GVL_1.Setpoint_M_Belts:=Setpoint_Belts_TOP_IN;
GVL_1.Setpoint_Belt_Feeder:=Setpoint_M_Belt_Feeder_IN;
GVL_1.Setpoint_SteamFan:=Setpoint_SteamFan_IN;
GVL_1.Setpoint_Compressor:=Setpoint_Compressor_IN;
GVL_1.Ps_202_out:=Ps_202;
GVL_1.Ps_203_out:=Ps_203;
GVL_1.volFracAir202_out:=volFracAir202;
GVL_1.volFracAir203_out:=volFracAir203;
GVL_1.volFracAirO2_out:=volFracAirO2;






IF SteamFAN_Switch_ON_manu AND SteamFan_ON_manu AND  Setpoint_SteamFan_Visu  >20.0 THEN
OK_For_HEAT_WHILE_FAN_IS_ON:=TRUE;
ELSE
OK_For_HEAT_WHILE_FAN_IS_ON:=FALSE;
END_IF;

END_PROGRAM

// ---- POUs/FB_Blink.TcPOU
FUNCTION_BLOCK FB_Blink
VAR_INPUT
	bStart:BOOL;
	tTakt:TIME:=t#0.5s;
END_VAR
VAR_OUTPUT
	bBlink:BOOL;
END_VAR
VAR
	fbT1:TON;
	fbT2:TON;
END_VAR

(*erste Hälfte der Blinkperiode, FB-Aufruf und Beschaltung in einem *)
fbT1(IN:=bStart AND NOT fbt2.Q,
	PT:= tTakt/2,
	Q=> bBlink,
	ET=> );


(*zweite Hälfte der Blinkperiode; Bsp. programmiert mit getrennter Beschaltung und Aufruf*)

fbt2.IN := fbT1.Q;   		(*vorheriges Beschalten der InputVar*)
fbt2.PT := tTakt / 2;  	(*vorheriges Beschalten der InputVar*)

fbT2();  					(*eigentliche FB-Instanz-Aufruf*)

END_FUNCTION_BLOCK

// ---- POUs/Average.TcPOU
FUNCTION_BLOCK Average
VAR_INPUT
	Input_AV: REAL;
END_VAR
VAR_OUTPUT
	OUTPUT_AV:REAL;
END_VAR
VAR
	C_AV: INT;
	summary_AV: REAL;
END_VAR



CASE C_AV OF


0:summary_AV:=0;	C_AV:=1;
1:summary_AV:=Input_AV;	C_AV:=2;
2:summary_AV:=summary_AV+Input_AV; C_AV:=3;
3:summary_AV:=summary_AV+Input_AV; C_AV:=4;
4:summary_AV:=summary_AV+Input_AV; C_AV:=5;
5:summary_AV:=summary_AV+Input_AV; C_AV:=6;
6:summary_AV:=summary_AV+Input_AV; C_AV:=7;
7:summary_AV:=summary_AV+Input_AV; C_AV:=8;
8:summary_AV:=summary_AV+Input_AV; C_AV:=9;
9:summary_AV:=summary_AV+Input_AV; C_AV:=10;
10:summary_AV:=summary_AV+Input_AV; C_AV:=11;
11:summary_AV:=summary_AV+Input_AV; C_AV:=12;
12:summary_AV:=summary_AV+Input_AV; C_AV:=13;
13:summary_AV:=summary_AV+Input_AV; C_AV:=14;
14:summary_AV:=summary_AV+Input_AV; C_AV:=15;
15:summary_AV:=summary_AV+Input_AV; C_AV:=16;
16:summary_AV:=summary_AV+Input_AV; C_AV:=17;
17:summary_AV:=summary_AV+Input_AV; C_AV:=18;
18:summary_AV:=summary_AV+Input_AV; C_AV:=19;
19:summary_AV:=summary_AV+Input_AV; C_AV:=20;
20:summary_AV:=summary_AV+Input_AV; C_AV:=21;
21:summary_AV:=summary_AV+Input_AV; C_AV:=22;
22:summary_AV:=summary_AV+Input_AV; C_AV:=23;
23:summary_AV:=summary_AV+Input_AV; C_AV:=24;
24:summary_AV:=summary_AV+Input_AV; C_AV:=25;
25:summary_AV:=summary_AV+Input_AV; C_AV:=26;
26:summary_AV:=summary_AV+Input_AV; C_AV:=27;
27:summary_AV:=summary_AV+Input_AV; C_AV:=28;
28:summary_AV:=summary_AV+Input_AV; C_AV:=29;
29:summary_AV:=summary_AV+Input_AV; C_AV:=30;
30:summary_AV:=summary_AV+Input_AV; C_AV:=31;
31:summary_AV:=summary_AV+Input_AV; C_AV:=32;
32:summary_AV:=summary_AV+Input_AV; C_AV:=33;
33:summary_AV:=summary_AV+Input_AV; C_AV:=34;
34:summary_AV:=summary_AV+Input_AV; C_AV:=35;
35:summary_AV:=summary_AV+Input_AV; C_AV:=36;
36:summary_AV:=summary_AV+Input_AV; C_AV:=37;
37:summary_AV:=summary_AV+Input_AV; C_AV:=38;
38:summary_AV:=summary_AV+Input_AV; C_AV:=39;
39:summary_AV:=summary_AV+Input_AV; C_AV:=40;
40:summary_AV:=summary_AV+Input_AV; C_AV:=41;
41:summary_AV:=summary_AV+Input_AV; C_AV:=42;
42:summary_AV:=summary_AV+Input_AV; C_AV:=43;
43:summary_AV:=summary_AV+Input_AV; C_AV:=44;
44:summary_AV:=summary_AV+Input_AV; C_AV:=45;
45:summary_AV:=summary_AV+Input_AV; C_AV:=46;
46:summary_AV:=summary_AV+Input_AV; C_AV:=47;
47:summary_AV:=summary_AV+Input_AV; C_AV:=48;
48:summary_AV:=summary_AV+Input_AV; C_AV:=49;
49:summary_AV:=summary_AV+Input_AV; C_AV:=50;
50:summary_AV:=summary_AV+Input_AV; C_AV:=51;
51:OUTPUT_AV:=summary_AV/50.0; C_AV:=0;

END_CASE

END_FUNCTION_BLOCK

// ---- POUs/Meine_HYST.TcPOU
FUNCTION_BLOCK Meine_HYST
VAR_INPUT
	Hyst_Value: INT;
	Hyst_Low_Limit: INT;
	Hyst_Hight_Limit: INT;
END_VAR
VAR_OUTPUT
	Hyst_OUT:BOOL ;
END_VAR
VAR
(*ZEITEN*)

	TON1:TON;
	IN_T1:BOOL;
	OUT_T1:BOOL;
	TON2:TON;
	IN_T2:BOOL;
	OUT_T2:BOOL;



END_VAR




(*Hyterese Universell für Heizmatten*)

IF Hyst_Value < Hyst_Low_Limit  THEN IN_T1:=TRUE; ELSE IF Hyst_Value  >= Hyst_Hight_Limit   THEN IN_T1:=FALSE; END_IF END_IF
IF OUT_T1 THEN Hyst_OUT:=TRUE; ELSE Hyst_OUT:=FALSE; END_IF



TON1(IN:=IN_T1 , PT:=t#30s, Q=>OUT_T1 , ET=> ); (*ZEIT Hauptschütz einschalten*)

TON2(IN:=IN_T2 , PT:=t#30s, Q=>OUT_T2 , ET=> ); (*ZEIT Überwachung Hauptschütz einschalten*)

END_FUNCTION_BLOCK

// ---- POUs/Controller.TcPOU
FUNCTION_BLOCK Controller
VAR_INPUT
END_VAR
VAR_OUTPUT
END_VAR
VAR
	CTRL_1: FB_BasicPID;
	CTRL_2: FB_BasicPID;
	
	Heat_REG1_CTRL:CTRL_PID;
	Heat_REG2_CTRL:CTRL_PID;
	Heat_REG3_CTRL:CTRL_PID;
	Heat_REG4_CTRL:CTRL_PID;
	Heat_REG5_CTRL:CTRL_PID;
	Heat_REG6_CTRL:CTRL_PID;
	Heat_REG7_CTRL:CTRL_PID;
	Heat_REG8_CTRL:CTRL_PID;
	
	
	
	Heat_REG1_PWM:CTRL_PWM;
	Heat_REG2_PWM:CTRL_PWM;
	Heat_REG3_PWM:CTRL_PWM;
	Heat_REG4_PWM:CTRL_PWM;
	Heat_REG5_PWM:CTRL_PWM;
	Heat_REG6_PWM:CTRL_PWM;
	Heat_REG7_PWM:CTRL_PWM;
	Heat_REG8_PWM:CTRL_PWM;
	
	
	
	
	
	fPWMDutyCycle1_out: REAL;
	fPWMDutyCycle2_out: REAL;
	fPWMDutyCycle3_out: REAL;
	fPWMDutyCycle4_out: REAL;
	
	
	
	
	
	HEAT_Reg_2_OUT_local: BOOL;
	HEAT_Reg_1_OUT_local: BOOL;
	HEAT_Reg_3_OUT_local: BOOL;
END_VAR





(* Infos zu den Reglern:

1. Es wurde eine von OSCAT-entwickelte Library-Sammlung zusammengefasst, damit diese auch als-FB/FC-Sammlung direkt im TC3-eingebunden werden können.
Die direkte Einbindung der OSCAT-Libs im Lib-Repository von TC3 macht Probleme, desshalb die direkte FB/FC Sammlung

In dieser Sammlung (Ornder PID_Controller_LIB) sind die CRT_PID & CTRL_PWM von OSCAT enthalten, welche für die Heizregler im Fall TRISS eingesetzt werden.

Wichtig als Backround: Die Controller_LIbs von Beckhoff sind etwas teuer, wenn nur die wesentlichen Grundfunktionen verwendet werden!!!

Andere Alternative wäre gewesen, wenn bei der Basic_PID Regler aus den Utility-Libs verwendet wird: (FB_BAsicPID) und selber eine umrechnung auf den PWM-Ausgang gemacht wird

Was sich nicht lohnt ist die Building-Automation LIB verwendet wird, da diese zwar einen Analog-PWM Ausgang beinhaltet, aber dieser PWM-Ausgang sehr "Primitiv" erstellt wurde

FAZIT: OSCAT so lange es geht & wenn dann zur Controller LIB von Beckhoff wechseln!!!
*)








	





	
	
(*

PID_CTRL

Type Funktionsbaustein
Input ACT : REAL (gemessener Wert nach der Strecke)
SET : REAL (Vorgabewert)
SUP : REAL (Rauschunterdrückung)
OFS : REAL (Ofset für den Ausgang)
M_I : REAL (Eingangswert für manuellen Betrieb)
MAN : BOOL (Umschalten auf Handbetrieb, MANUAL = TRUE)
RST : BOOL (Asynchroner Reset-Eingang)
KP : REAL (Verstärkung des Reglers)
TN : REAL (Nachstellzeit des Reglers)
TV : REAL (Vorhaltezeit des Reglers)
LL : REAL (untere Ausgangsbegrenzung)
LH : REAL (obere Ausgangsbegrenzung)
Output Y : REAL (Ausgang des Reglers)
DIFF : Real (Regelabweichung)
LIM : BOOL (TRUE, wenn der Ausgang ein Limit erreicht hat)


CTRL_PID ist ein PID-Regler mit dynamischen Anti Wind-Up und manuellem
Steuereingang. Der PID Regler arbeitet nach der Formel:
Y = KP * ( DIFF + 1/TN * INTEG(DIFF) + TV *DERIV(DIFF)) + OFFSET
wobei DIFF = SET_POINT – ACTUAL
Im Handbetrieb (Manual = TRUE) gilt: Y = MANUAL_IN + OFFSET
ACT ist der gemessene Wert nach der Regelstrecke und SET ist die Sollwertvorgabe
für den Regler. Die Eingangswerte LH und LL begrenzen den
Ausgangswert Y. Mit RST kann der interne Integrator jederzeit auf 0 gesetzt
werden. Der Ausgang LIM signalisiert das der Regler an eine der
Grenzen LL oder LH gelaufen ist. Der PID-Regler arbeitet frei laufend und
benutzt zur Berechnung die Trapezregel für höchste Genauigkeit und optimale
Geschwindigkeit. Die Default-Werte der Eingangsparameter sind wie
folgt vordefniert: KP = 1, TN = 1, TV = 1, LIMIT_L = -1000 und LIMIT_H =
+1000. Mit dem Eingang SUP wird eine Rauschunterdrückung eingestellt,
der Wert am Eingang SUP legt fest ab welcher Regeldiferenz der Regler
einschaltet. Mit SUP wird vermieden das der Ausgang des Reglers dauern
schwankt. Der Wert am Eingang SUP sollte so bemessen sein das er das
Rauschen der Regelstrecke und der Sensoren unterdrückt. Wird zum Beispiel
der Eingang SUP auf 0.1 gesetzt so wird der Regler erst bei Regelabweichungen
größer als 0.1 aktiv. Der Ausgang DIFF stellt die gemessene
und durch ein Noise Filter (DEAD_BAND) geflterte Regelabweichung zur
Verfügung. DIFF wird in einer Regelstrecke normalerweise nicht benötigt,
kann aber zur Beeinfussung der Regelparameter benutzt werden. Der Eingang
OFS wird als letzter Wert zum Ausgang addiert, und dient vor allem
zum kompensieren von Störsignalen, deren Wirkung auf den Regelkreis
abgeschätzt werden kann.
Der Regler arbeitet mit einem Dynamischen Wind-Up das verhindert dass
der Integrator bei erreichen eines Ausgangslimits und weiterer Regelabweichung
unbegrenzt weiter läuft und die Regeleigenschaften negativ beeinfusst.
In der Einleitung des Kapitel Regelungstechnik fnden sich weitere
Details zum Thema Anti Wind-Up.





PWM:
CTRL_PWM
Type Funktionsbaustein
Input CI : REAL (Eingang vom Controller)
MAN_IN : REAL (Manueller Eingangswert)
MANUAL : BOOL (Umschalter für Handbetrieb)
F : REAL (Frequenz der Ausgangsimpulse in Hz)
Output Q : BOOL (Steuersignal)


CTRL_PWM wandelt den Eingangswert CI (0..1) in ein Pulsweitenmoduliertes
Ausgangssignal Q. Wenn MANUAL = TRUE wird am Ausgang Q Der Eingangswert
von MAN_IN ausgegeben. CTRL_OUT kann benutzt werden um
eigene Regelbausteine Aufzubauen.
397
*)









//Verknüpfung = PID Regler => PWM => OUTPUT
	
//Heizregister Gruppe 1 oben 1-4


Heat_reg1_CTRL(
	ACT:=T_Einduesung_oben_Visu , 
	SET:=fSetpointValue1 , 
	SUP:= , 
	OFS:= , 
	M_I:= , 
	MAN:= , 
	RST:= , 
	KP:=fKP_Controller_Heatmatt1 , 
	TN:=fKI_Controller_Heatmatt1, 
	TV:= 0.1 , 
	LL:= 0, 
	LH:= 100, 
	Y=>fPWMDutyCycle1 , 
	DIFF=> , 
	LIM=> );


fPWMDutyCycle1_out:=(fPWMDutyCycle1/100)*1;

Heat_reg1_PWM(
	CI:= fPWMDutyCycle1_out, 
	MAN_IN:= , 
	MANUAL:= , 
	F:=1 , 
	Q=> bAuto_Heat_REG1_CTRL);


	



	
	

	
	
	
	
	
	//Heizregister Gruppe 2 unten 5-8

Heat_reg2_CTRL(
	ACT:=T_Einduesung_unten_Visu , 
	SET:=fSetpointValue2 , 
	SUP:= , 
	OFS:= , 
	M_I:= , 
	MAN:= , 
	RST:= , 
	KP:=fKP_Controller_Heatmatt2 , 
	TN:=fKI_Controller_Heatmatt2, 
	TV:= 0.1 , 
	LL:= 0, 
	LH:= 100, 
	Y=>fPWMDutyCycle2 , 
	DIFF=> , 
	LIM=> );


fPWMDutyCycle2_out:=(fPWMDutyCycle2/100)*1;

Heat_reg2_PWM(
	CI:= fPWMDutyCycle2_out, 
	MAN_IN:= , 
	MANUAL:= , 
	F:=1 , 
	Q=> bAuto_Heat_REG2_CTRL );


	
	
	
	
	
	
//Heizregister bei Kompressor (verhinderung von Kondensation)




Heat_reg3_CTRL(
	ACT:=T_Komp_Gehaeuse_Visu , 
	SET:=fSetpointValue3 , 
	SUP:= , 
	OFS:= , 
	M_I:= , 
	MAN:= , 
	RST:= , 
	KP:=fKP_Controller_Heatmatt3 , 
	TN:=fKI_Controller_Heatmatt3, 
	TV:= 0.1 , 
	LL:= 0, 
	LH:= 100, 
	Y=>fPWMDutyCycle3 , 
	DIFF=> , 
	LIM=> );


fPWMDutyCycle3_out:=(fPWMDutyCycle3/100)*1;

Heat_reg3_PWM(
	CI:= fPWMDutyCycle3_out, 
	MAN_IN:= , 
	MANUAL:= , 
	F:=1 , 
	Q=> bAuto_Heat_REG3_CTRL);
	
	

	
	
	
	HEAT_Reg_1_OUT:=HEAT_Reg_1_OUT_local;
	HEAT_Reg_2_OUT:=HEAT_Reg_2_OUT_local;
	HEAT_Reg_3_OUT:=HEAT_Reg_3_OUT_local;
	HEAT_Reg_4_OUT:=HEAT_Reg_4_manu;
	HEAT_Reg_5_OUT:=HEAT_Reg_5_manu;
	HEAT_Reg_6_OUT:=HEAT_Reg_6_manu;
	HEAT_Reg_7_OUT:=HEAT_Reg_7_manu;
	HEAT_Reg_8_OUT:=HEAT_Reg_8_manu;


	HEAT_Reg_Mainswitch_out:=HEAT_Reg_Mainswitch_manu;

	
	
	
	
	
	
	
	


(* Der Regler soll vorübergehend so funktionieren, dass im Haupt-Manu Mode der regeler im Auto-Modus läuft*)
	IF Ctr_Manu AND Control_Manu_active =FALSE THEN

	 Ctr_Manu_active:=TRUE;
	 Ctr_Auto_active:=FALSE;
	 Ctr_Reset_active:=FALSE;
	ELSE IF Control_Manu_active THEN
	
	 Ctr_Manu_active:=FALSE;
	 Ctr_Auto_active:=TRUE;
	 Ctr_Reset_active:=FALSE;
	ELSE IF Ctr_Reset THEN
	 Ctr_Manu_active:=FALSE;
	 Ctr_Auto_active:=FALSE;
	 Ctr_Reset_active:=TRUE;
	
	END_IF
	END_IF
	END_IF



	
	

(*Wichtige info: Zurzeit  ist der Manu-Ausgang der Haupt-Ausgang, auch wenn der Regler im Auto_Modus arbeitet*)



//Regler Heizregister 1-4 und 5-8

IF T_HE_Einduesung_Oben_Visu > T_Limit_Heatreg_top  OR 
fTemp_mean_belt_top > T_Limit_Heatreg_top OR
OK_For_HEAT_WHILE_FAN_IS_ON = FALSE OR
bManuHeat_REG1_switch_ON = FALSE THEN
HEAT_Reg_1_Manu:=FALSE;
bAuto_Heat_REG1_CTRL:=FALSE;
HEAT_Reg_1_OUT:=FALSE;
//HEAT_Reg_1_auto:=FALSE;
ELSE
HEAT_Reg_1_OUT_local:=bManuHeat_REG1_CTRL OR bAuto_Heat_REG1_CTRL;
END_IF;



IF T_HE_Einduesung_unten_Visu > T_Limit_Heatreg_bottom  OR 
fTemp_mean_belt_bottom > T_Limit_Heatreg_bottom OR
OK_For_HEAT_WHILE_FAN_IS_ON = FALSE  OR  
bManuHeat_REG2_switch_ON = FALSE THEN
HEAT_Reg_2_OUT:=FALSE;
bAuto_Heat_REG2_CTRL:=FALSE;
HEAT_Reg_2_OUT:=FALSE;
//HEAT_Reg_2_auto:=FALSE;
ELSE
HEAT_Reg_2_OUT_local:=bManuHeat_REG2_CTRL OR bAuto_Heat_REG2_CTRL;
END_IF;



//OK_For_HEAT_WHILE_FAN_IS_ON:=SteamFAN_Switch_ON_manu AND SteamFan_ON_manu AND Setpoint_SteamFan_Visu >=0;

//Versuch mal so, wiel Preobleme mit Zeile oben:
IF SteamFAN_Switch_ON_manu AND SteamFan_ON_manu AND Setpoint_SteamFan_Visu >= 20.0 THEN
OK_For_HEAT_WHILE_FAN_IS_ON:=TRUE;
ELSE
OK_For_HEAT_WHILE_FAN_IS_ON:=FALSE;
END_IF;



//Heizregister bei Kompressor (verhinderung von Kondensation)


IF  T_Komp_Gehaeuse_Visu > T_Limit_Heatreg3  OR  bManuHeat_REG3_switch_ON = FALSE THEN

HEAT_Reg_3_OUT:=FALSE;
bAuto_Heat_REG3_CTRL:=FALSE;
HEAT_Reg_3_OUT:=FALSE;
//HEAT_Reg_3_auto:=FALSE;

ELSE
	
HEAT_Reg_3_OUT_local:=bManuHeat_REG3_CTRL OR bAuto_Heat_REG3_CTRL;


END_IF;






	(*Hier wird der Setpoint automatisch auf 0 gesetzt*)



	IF  Main_Relais = FALSE THEN
		
	bManuHeat_REG1_CTRL:=FALSE;
	bManuHeat_REG2_CTRL:=FALSE;
	bManuHeat_REG3_CTRL:=FALSE;
	bManuHeat_REG4_CTRL:=FALSE;
	
	bAuto_Heat_REG1_CTRL:=FALSE;
	bAuto_Heat_REG2_CTRL:=FALSE;
	bAuto_Heat_REG3_CTRL:=FALSE;
	bAuto_Heat_REG4_CTRL:=FALSE;
	
	fSetpointValue1:=0;
	fSetpointValue2:=0;
	fSetpointValue3:=0;
	fSetpointValue4:=0;
	
	
	END_IF;








fTemp_mean_belt_top:= (T_HE_Einduesung_oben_Visu + T_Einduesung_oben_Visu) /2.0;

fTemp_mean_belt_bottom:= (T_HE_Einduesung_Unten_Visu + T_Einduesung_Unten_Visu) /2.0;

END_FUNCTION_BLOCK

// ---- POUs/Control_LIbs/CTRL_PID.TcPOU
FUNCTION_BLOCK CTRL_PID
VAR_INPUT
	ACT, SET, SUP, OFS, M_I : REAL;
	MAN : BOOL;
	RST : BOOL;
	KP : REAL := 1.0;
	TN : REAL := 1.0;
	TV : REAL := 1.0;
	LL : REAL := -1000.0;
	LH : REAL := 1000.0;
END_VAR
VAR_OUTPUT
	Y : REAL;
	DIFF : REAL;
	LIM : BOOL;
END_VAR
VAR
	pid : FT_PIDWL;
	co : CTRL_OUT;
END_VAR



(*
version 2.0	30. jun. 2008
programmer 	hugo
tested by	oscat

FT_PI is a PI controller with manual functionality.
The PID controller works according to the fomula Y = e *(KP+ KI * INTEG(e) ) + offset, while e = set_point - actual.
a rst will reset all internal data, while a switch to manual will cause the controller to follow the function Y = manual_in + offset.
limit_h and Limit_l set the possible output range of Y.
the output flags lim will signal that the output limits are active.

*)

DIFF := CTRL_IN(SET, ACT, SUP);
pid(in := DIFF, kp := KP, tn := TN, tv := TV, lim_l := LL, lim_h := LH, rst := RST);
co(ci := pid.Y, OFFSET := OFS, man_in := M_I, lim_l := LL, lim_h := LH, MANUAL := MAN);
Y := co.Y;
LIM := co.LIM;



(* revision history

hm 1.12.2006	 	rev 1.1
	changed algorithm to trapezregel for higher accuracy.

hm 3.1.2007		rev 1.2
	added integ_band to select when the integrator is active.

hm	3.3.2007		rev 1.3
	added default values to inputs KP, TN, TV, LIMIT_L und LIMIT_H.

hm 31.oct 2007	rev 1.4
	total rewrite of the module to avoid failures when one of the limits is 0

hm	3.11.2007	rev 1.5
	added noise input to filter noise
	added output diff
	set limit output false when output is within limits
	overfolw was not set correctly

hm	5. jan 2008	rev 1.6
	improved code for better performance
*)

END_FUNCTION_BLOCK

// ---- POUs/Control_LIbs/FT_PIDWL.TcPOU
FUNCTION_BLOCK FT_PIDWL
VAR_INPUT
	IN : REAL;
	KP : REAL := 1.0;
	TN : REAL := 1.0;
	TV : REAL := 1.0;
	LIM_L : REAL := -1.0E38;
	LIM_H : REAL := 1.0E38;
	RST : BOOL;
END_VAR
VAR_OUTPUT
	Y : REAL;
	LIM : BOOL;
END_VAR
VAR
	piwl : FT_PIWL;
	diff : FT_DERIV;
END_VAR

(*
version 1.3	13. nov. 2009
programmer 	hugo
tested by		tobias

FT_PIDWL is a PID controller with dynamic wind_up reset.
The PID controller works according to the fomula Y = KP *(IN + KI * INTEG(e) + DERIV(e) ).
a rst will reset the integrator to 0
lim_h and Lim_l set the possible output range of the internal integrator.
the output flags lim will signal that the output limits are active.

default values for KP = 1, KI = 1, ILIM_L = -1E37, iLIM_H = +1E38.
*)

(* if rst then *)
IF rst THEN
	piwl(rst := TRUE);
	piwl.RST := FALSE;
ELSE
	(* run PIWL controller first *)
	(* we need to check if TN = 0 and do alternative calls *)
	IF TN = 0.0 THEN
		piwl(in := IN * KP, KP := 1.0, KI := 0.0, LIM_L := LIM_L, LIM_H := LIM_H);
	ELSE
		piwl(in := IN * KP, KP := 1.0, KI := 1.0 / TN, LIM_L := LIM_L, LIM_H := LIM_H);
	END_IF;

	(* run differentiator and add_to_output *)
	diff(IN := IN, K := KP * TV);
	Y := piwl.Y + diff.out;

	(* limit the output *)
	IF Y < LIM_L THEN
		LIM := TRUE;
		Y := LIM_L;
	ELSIF Y > LIM_H THEN
		LIM := TRUE;
		Y := LIM_H;
	ELSE
		LIM := FALSE;
	END_IF;
END_IF;



(* revision history
hm 13. jun. 2008 	rev 1.0
	original version

hm	25. jan 2008	rev 1.1
	multiply differential part with KP

hm	11. mar. 2009	rev 1.2
	real constants updated to new systax using dot

hm	13. nov. 2009	rev 1.3
	fixed code for negative KP

*)

END_FUNCTION_BLOCK

// ---- POUs/Control_LIbs/FT_PIWL.TcPOU
FUNCTION_BLOCK FT_PIWL
VAR_INPUT
	IN : REAL;
	KP : REAL := 1.0;
	KI : REAL := 1.0;
	LIM_L : REAL := -1.0E38;
	LIM_H : REAL := 1.0E38;
	RST : BOOL;
END_VAR
VAR_OUTPUT
	Y : REAL;
	LIM : BOOL;
END_VAR
VAR
	init: BOOL;
	tx: DWORD;
	tc : REAL;
	t_last: DWORD;
	in_last : REAL;
	i: REAL;
	p: REAL;
END_VAR

(*
version 1.3	11. mar. 2009
programmer 	hugo
tested by		oscat

FT_PIWL is a PI controller.
The PID controller works according to the fomula Y = IN *(KP+ KI * INTEG(e) ).
a rst will reset the integrator to 0
lim_h and Lim_l set the possible output range of the controller.
the output flag lim will signal that the output limits are active.
the integrator ist equipped with anti wind-up circuitry which limits trhe total output ranke to lim_l and lim_h

default values for KP = 1, KI = 1, ILIM_L = -1E37, iLIM_H = +1E38.
*)

(* initialize at power_up *)
IF NOT init OR RST THEN
	init := TRUE;
	in_last := in;
	t_last := T_PLC_US();
	i := 0.0;
	tc := 0.0;
ELSE
	(* read last cycle time in Microseconds *)
	tx := T_PLC_US();
	tc := DWORD_TO_REAL(tx - t_last);
	t_last := tx;

	(* calculate proportional part *)
	p := KP * IN;

	(* run integrator *)
	i := (IN + in_last) * 5.0E-7 * KI * tc + i;
	in_last := IN;

	(* calculate output Y *)
	Y := p + i;

	(* check output for limits *)
	IF Y >= LIM_H THEN
		Y := LIM_H;
		IF ki <> 0.0 THEN
			i := LIM_H - p;
		ELSE
			i := 0.0;
		END_IF;
		LIM := TRUE;
	ELSIF Y <= LIM_L THEN
		Y := LIM_L;
		IF ki <> 0.0 THEN
			i := LIM_L - p;
		ELSE
			i := 0.0;
		END_IF;
		LIM := TRUE;
	ELSE
		LIM := FALSE;
	END_IF;
END_IF;




(* revision history
hm 13. jun. 2008 	rev 1.0
	original version

hm	27. oct. 2008	rev 1.1
	integrator will not be adjusted when ki = 0

hm	25. jan 2009	rev 1.2
	module will also work with negative K

hm	11. mar. 2009	rev 1.3
	real constants updated to new systax using dot

*)

END_FUNCTION_BLOCK

// ---- POUs/Control_LIbs/T_PLC_US.TcPOU
FUNCTION T_PLC_US : DWORD
VAR CONSTANT
	debug : BOOL := 0;
	N : INT := 0;
	offset : DWORD := 0;
END_VAR
VAR
	tx : TIME;
END_VAR

(*
version 1.2	16 nov 2008
programmer 	hugo
tested by	tobias

T_PLC_US reads the internal PLC timer and return the time, it has the advantage to be able to set a debug mode 
and speed up the counter to test the plc timer overrun which occurs every 50 days respectively 25 days at siemens S7
this routine also allows to correct the behavior of s7 where the internal plc counter will not count all 32 bits.

*)

tx := TIME();
T_PLC_US := TIME_TO_DWORD(Tx)*1000;
(* hier muss die korrektur für step7 stattfinden
plctime muss den vollen wertebereich von time ausnutzen:
wenn bei step7 time -24tage bis plus 24 tage ist dann muss der timer auch beim überlauf auf -24tage springen 
und auf keinen fall auf 0 !!!!
für siemens muss ein weiterer fb im main eingebunden werden der sicherstellt das alle 32 bits durchgezählt werden.
es kann nur ein fb sein den er muss sich das oberste (32te) bit merken.
oder etwa spring s7 bei überlauf auf -24 tage????? dann wäre keine korrektur nötig.
*)
IF debug THEN
	T_PLC_US := (SHL(T_PLC_US,N) OR SHL(DWORD#1,N)-1) + OFFSET;
END_IF;

(* revision history
hm	14.9.2007	rev 1.0
	original version

hm	12. nov 2007	rev 1.1
	added temporaray variable tx because some compilers could not handle time() as an argument

hm	16. nov. 2008	rev 1.2
	initialized constants with 0 for compatibility reasons

*)

END_FUNCTION

// ---- POUs/Control_LIbs/FT_DERIV.TcPOU
FUNCTION_BLOCK FT_DERIV
VAR_INPUT
	in : REAL;
	K : REAL := 1.0;
	run : BOOL := TRUE;
END_VAR
VAR_OUTPUT
	out : REAL;
END_VAR
VAR
	old: REAL;
	tx: DWORD;
	last: DWORD;
	init: BOOL;
	tc: REAL;
END_VAR


(*
version 1.5	11. mar. 2009
programmer 	hugo
tested by		oscat

FT_deriv calculates the derivate over the signal "in" with Faktor "K".
a run input enables or stops the calculation, if left unconnected its true and therfore the calculation is executed.
if K is not specified the default is 1.

*)

(* read system time *)
tx := T_PLC_US();
tc := DWORD_TO_REAL(tx - last);
last := tx;

(* init on first startup *)
IF NOT init THEN
	init := TRUE;
	old := in;
ELSIF run AND tc > 0.0 THEN
	out := (in - old) / tc * 1000000.0 * K;
	old := in;
ELSE
	out := 0.0;
END_IF;



(*
hm 3.1.2007			rev 1.1
	added init code for startup
	set the default for K to 1

hm	15. sep 2007	rev 1.2
	replaced Time() with T_PLC_US for compatibility and performance reasons
	increased accuracy and work in microseconds internally

hm 29 oct 2007	rev 1.3
	prohibit calculation when tx - last = 0 to avoid division by 0 and increase accuracy on fast systems

hm	6. nov. 2008	rev 1.4
	improved performance

hm	11. mar. 2009	rev 1.5
	inproved code
*)

END_FUNCTION_BLOCK

// ---- POUs/Control_LIbs/CTRL_OUT.TcPOU
FUNCTION_BLOCK CTRL_OUT
VAR_INPUT
	CI, OFFSET, MAN_IN, LIM_L, LIM_H : REAL;
	MANUAL : BOOL;
END_VAR
VAR_OUTPUT
	Y : REAL;
	LIM : BOOL;
END_VAR


(*
version 1.1	5. nov 2008
programmer 	hugo
tested by	oscat


*)

Y := SEL(MANUAL, CI, MAN_IN) + OFFSET;

(* Limit the output *)
IF Y > LIM_L AND Y < LIM_H THEN
	LIM := FALSE;
ELSE
	Y := LIMIT(LIM_L, Y, LIM_H);
	LIM := TRUE;
END_IF;



(* revision history
hm 	2. jun. 2008 	rev 1.0
	original version

hm	5. nov. 2008	rev 1.1
	optimized code
*)

END_FUNCTION_BLOCK

// ---- POUs/Control_LIbs/CTRL_IN.TcPOU
FUNCTION CTRL_IN : REAL
VAR_INPUT
	SET_POINT, ACTUAL, NOISE : REAL;
END_VAR


(*
version 1.0	2. jun 2008
programmer 	hugo
tested by		tobias


*)

(* calculate the process error DIFF *)
CTRL_IN := DEAD_ZONE(SET_POINT - ACTUAL, NOISE);


(* revision history
hm 	2. jun. 2008 	rev 1.0
	original version

*)

END_FUNCTION

// ---- POUs/Control_LIbs/DEAD_ZONE.TcPOU
FUNCTION DEAD_ZONE : REAL
VAR_INPUT
	X : REAL;
	L : REAL;
END_VAR


(*
version 1.2	11. mar. 2009
programmer 	hugo
tested by		oscat

dead_zone2 is a linear transfer function which follows a linear function except for x is close to 0.
Y = X if abs(x) > L otherwise its 0.

*)

IF ABS(x) > L THEN
	dead_zone := X;
ELSE
	DEAD_ZONE := 0.0;
END_IF;

(* revision history
hm	12. feb. 2007	rev 1.0
	original version

hm	14. jun. 2008	rev 1.1
	improved performance

hm	11. mar. 2009	rev 1.2
	real constants updated to new systax using dot

*)

END_FUNCTION

// ---- POUs/Control_LIbs/CTRL_PWM.TcPOU
FUNCTION_BLOCK CTRL_PWM
VAR_INPUT
	CI, MAN_IN : REAL;
	MANUAL : BOOL;
	F : REAL;
END_VAR
VAR_OUTPUT
	Q : BOOL;
END_VAR
VAR
	PW : PWM_DC;
END_VAR

(*
version 1.1	21. oct. 2008
programmer 	hugo
tested by	oscat


*)

PW(F := F, DC := SEL(MANUAL,CI,MAN_IN));
Q := PW.Q;


(* revision history
hm 3. jun. 2008 	rev 1.0
	original version

hm	21. oct. 2008	rev 1.1
	optimized code

*)

END_FUNCTION_BLOCK

// ---- POUs/Control_LIbs/PWM_DC.TcPOU
FUNCTION_BLOCK PWM_DC
VAR_INPUT
	F : REAL;
	DC : REAL;
END_VAR
VAR_OUTPUT
	Q : BOOL;
END_VAR
VAR
	clk: CLK_PRG;
	pulse: TP_X;
	tmp: REAL;
END_VAR

(*
version 1.4	11. mar. 2009
programmer 	oscat
tested BY		oscat

this signal generator generates a square wave signal which is specified by the frequency and the duty cycle
*)

IF F > 0.0 THEN
	tmp := 1000.0 / F;
	CLK(PT := REAL_TO_TIME(tmp));
	Pulse(in := clk.Q, pt := REAL_TO_TIME(tmp * DC));
	Q := pulse.Q;
END_IF;

(* revision history

hm	25. feb 2007	rev 1.1
	recoded in st for better performance and better portability

hm	27. nov 2007	rev 1.2
	avoid divide by 0 when F = 0

hm	19. oct. 2008	rev 1.3
	changed type TP_R to TP_X because of name change
	improved performance

hm	11. mar. 2009	rev 1.4
	changed real constants to use dot syntax

*)

END_FUNCTION_BLOCK

// ---- POUs/Control_LIbs/CLK_PRG.TcPOU
	FUNCTION_BLOCK CLK_PRG
VAR_INPUT
	PT : TIME := t#10ms;
END_VAR
VAR_OUTPUT
	Q : BOOL;
END_VAR
VAR
	init : BOOL;
	last : TIME;
	tx: TIME;
END_VAR

(*
version 1.3	25. oct. 2008
programmer 	hugo
tested by		tobias

clk_prg uses the internal sps time to generate a clock with programmable period time.
the first cycle after start is a clk pulse and then depending on the programmed period time a delay.
every pulse is only valid for one cycle.
the accuracy of clk_prg is depending on the accuracy of the system clock.

*)

(* read system time *)
tx := DWORD_TO_TIME(T_PLC_MS());

(* initialize on startup *)
IF NOT init THEN
	init := TRUE;
	last := tx - pt;
END_IF;

(* generate output pulse when next_pulse is reached *)
Q := tx - last >= pt;
IF Q THEN last := tx; END_IF;


(* revision hiostory

hm 25 feb 2007	rev 1.1
	rewritten code for higher performance
	pt can now be changed during runtime

hm	17. sep 2007	rev 1.2
	replaced time() with t_plc_ms() for compatibility reasons

hm	25. oct. 2008	rev 1.3
	optimized code

*)

END_FUNCTION_BLOCK

// ---- POUs/Control_LIbs/T_PLC_MS.TcPOU
FUNCTION T_PLC_MS : DWORD
VAR CONSTANT
	debug : BOOL := 0;
	N : INT := 0;
	offset : DWORD := 0;
END_VAR
VAR
	tx : TIME;
END_VAR

(*
version 1.2	16. nov 2008
programmer 	hugo
tested by	oscat

T_PLC_MS reads the internal PLC timer and return the time, it has the advantage to be able to set a debug mode 
and speed up the counter to test the plc timer overrun which occurs every 50 days respectively 25 days at siemens S7
this routine also allows to correct the behavior of s7 where the internal plc counter will not count all 32 bits.

*)

tx := TIME();
T_PLC_MS := TIME_TO_DWORD(Tx);
(* hier muss die korrektur für step7 stattfinden
plctime muss den vollen wertebereich von time ausnutzen:
wenn bei step7 time -24tage bis plus 24 tage ist dann muss der timer auch beim überlauf auf -24tage springen 
und auf keinen fall auf 0 !!!!
für siemens muss ein weiterer fb im main eingebunden werden der sicherstellt das alle 32 bits durchgezählt werden.
es kann nur ein fb sein den er muss sich das oberste (32te) bit merken.
oder etwa spring s7 bei überlauf auf -24 tage????? dann wäre keine korrektur nötig.
*)
IF debug THEN
	T_PLC_MS := (SHL(T_PLC_MS,N) OR SHL(DWORD#1,N)-1) + OFFSET;
END_IF;

(* revision history
hm	14.9.2007	rev 1.0
	original version

hm	12. nov 2007	rev 1.1
	added temporaray variable tx because some compilers could not handle time() as an argument

hm	16. nov. 2008	rev 1.2
	initialized constants with 0 for compatibility reasons
*)

END_FUNCTION

// ---- POUs/Control_LIbs/TP_X.TcPOU
FUNCTION_BLOCK TP_X
VAR_INPUT
	IN : BOOL;
	PT : TIME;
END_VAR
VAR_OUTPUT
	Q : BOOL;
	ET : TIME;
END_VAR
VAR
	edge : BOOL;
	start : TIME;
	tx: TIME;
END_VAR

(*
version 1.3	17. dec. 2008
programmer 	hugo
tested by	oscat

retriggerable edge triggered pulse similar to TP but with a retrigger function
if the pt input is 0 then output is always low.
*)

(* read system_time *)
tx := DWORD_TO_TIME(T_PLC_MS());

(* rising edge trigger *)
IF IN AND NOT edge THEN
	start := tx;
	Q := PT > t#0ms;
ELSIF Q THEN
	ET := tx - start;
	IF ET >= PT THEN
		Q := FALSE;
		ET := t#0ms;
	END_IF;
END_IF;
edge := IN;

(* revision history
hm	4. aug 2006		rev 1.0
	original version

hm	17. sep 2007	rev 1.1
	replaced time() with T_PLC_MS() for compatibility reasons

hm	19. oct. 2008	rev 1.2
	renamed to TP_R to TP_X for compatibility reasons

hm	17. dec. 2008	rev 1.3
	code optimized

*)

END_FUNCTION_BLOCK

// ---- POUs/FB_PeerToPeer.TcPOU
(* Function block example of UDP peer-to-peer application *)
FUNCTION_BLOCK FB_PeerToPeer
VAR_IN_OUT
	fbTx		: FB_FrameFifo;(* TX fifo *)
	fbRx		: FB_FrameFifo;(* RX fifo *)
	fbLog		: FB_LogFifo;(* Log message fifo *)
END_VAR
VAR_INPUT
	sSrvNetId		: T_AmsNetID 	:= '';(* TwinCAT TCP/IP server network address. Default: empty string. *)
	sLocalHost		: T_IPv4Addr 	:= '192.168.100.88';(* Local address: String containing an (Ipv4) Internet Protocol dotted address. *)
	nLocalPort		: UDINT 		:= 0;(* Local address: IP port number. *)
	bEnable 		: BOOL			:= true;(* TRUE => Enable/connect, FALSE => Disable/disconnect *)
	tReconnect		: TIME			:= T#5S;(* Reconnect delay time *)
	bLog			: BOOL			:= FALSE;(* TRUE => Enable log message output, FALSE => Disable *)
	sPrefix			: STRING 		:= 'PeerToPeerX::';(* Log message description string (allows the identification of log message source) *)
END_VAR
VAR_OUTPUT
	bCreated		: BOOL;(* Connectionless socket state (TRUE => created, FALSE => closed) *)
END_VAR
VAR
	fbCreate		: FB_SocketUdpCreate;
	fbClose			: FB_SocketClose;
	fbReceiveFrom	: FB_SocketUdpReceiveFrom;
	fbSendTo		: FB_SocketUdpSendTo;
	stSendTo		: ST_FrameFifoEntry;
	stReceivedFrom	: ST_FrameFifoEntry;
	fbCreateTimer	: TON := ( PT := T#0S );	
	eStep			: E_ClientServerSteps;
END_VAR



//für ehemals test mit IAS kann die UPD kommunikation verwendet werden!


(*

CASE eStep OF
	eUDP_STATE_IDLE:
		IF bEnable XOR bCreated THEN
			IF bEnable THEN
				fbTx.Clear( sPrefix := CONCAT( sPrefix, 'FB_FrameFifo(sender)::' ), bLog := bLog );(* Clear send fifo *)
				fbRx.Clear( sPrefix := CONCAT( sPrefix, 'FB_FrameFifo(receiver)::' ), bLog := bLog );(* Clear receiver fifo *)
				fbLog.Clear( sPrefix := sPrefix, bLog := bLog );(* Clear log fifo *)

				(* At program start (first time) connect emmediately, next time after delay time *)
				fbCreateTimer( IN := TRUE );
				IF fbCreateTimer.Q THEN
					fbCreateTimer( IN := FALSE, PT := tReconnect ); 
					eStep := eUDP_STATE_CREATE_START;
				END_IF
			
			ELSE
				eStep := eUDP_STATE_CLOSE_START;
			END_IF
		ELSIF bCreated THEN
			fbTx.RemoveHead( stGet => stSendTo );
			IF fbTx.bOk THEN
				eStep := eUDP_STATE_SEND_START;
			ELSE (* Empty *)
				eStep := eUDP_STATE_RECEIVE_START;
			END_IF
		ELSE
			fbCreateTimer( IN := FALSE, PT := T#0S );
		END_IF

	eUDP_STATE_CREATE_START:
		fbCreate( bExecute := FALSE  );
		fbCreate( sSrvNetId := sSrvNetId, sLocalHost:= sLocalHost, nLocalPort:= nLocalPort, bExecute:= TRUE );
		eStep := eUDP_STATE_CREATE_WAIT;

	eUDP_STATE_CREATE_WAIT:
		fbCreate( bExecute := FALSE );
		IF NOT fbCreate.bBusy THEN
			IF NOT fbCreate.bError THEN
				bCreated := TRUE;
				fbLog.Message( sMessage := 'Connectionless (UDP) socket created!', hSocket := fbCreate.hSocket );
				eStep := eUDP_STATE_IDLE;
			ELSE
				fbLog.Error( sMessage := 'FB_SocketUdpCreate()', nErrID := fbCreate.nErrID );
				eStep := eUDP_STATE_ERROR;
			END_IF
		END_IF

	eUDP_STATE_SEND_START:
		fbSendTo( bExecute := FALSE );
		fbSendTo( sSrvNetId := sSrvNetId, sRemoteHost := stSendTo.stRemoteAddr.sAddr,
					nRemotePort := stSendTo.stRemoteAddr.nPort,
					pSrc:= ADR( stSendTo.sMessage ),
					cbLen:= INT_TO_UDINT(LEN( stSendTo.sMessage )) + 1, (* Include the end delimiter *)
					hSocket:= fbCreate.hSocket, bExecute:= TRUE );
		eStep := eUDP_STATE_SEND_WAIT;

	eUDP_STATE_SEND_WAIT:
		fbSendTo( bExecute := FALSE );
		IF NOT fbSendTo.bBusy THEN
			IF NOT fbSendTo.bError THEN
				eStep := eUDP_STATE_RECEIVE_START;
			ELSE
				fbLog.Error( sMessage := 'FB_SocketUdpSendTo()', nErrID := fbSendTo.nErrID );
				eStep := eUDP_STATE_ERROR;
			END_IF
		END_IF

	eUDP_STATE_RECEIVE_START:
		MEMSET( ADR( stReceivedFrom ), 0, SIZEOF( stReceivedFrom ) );
		fbReceiveFrom( bExecute := FALSE );
		fbReceiveFrom( sSrvNetId := sSrvNetId, 
						pDest:= ADR( stReceivedFrom.sMessage ),
						cbLen:= SIZEOF( stReceivedFrom.sMessage ) - 1, (* Without string delimiter *)
						hSocket:= fbCreate.hSocket, bExecute:= TRUE );
		eStep := eUDP_STATE_RECEIVE_WAIT;

	eUDP_STATE_RECEIVE_WAIT:
		fbReceiveFrom( bExecute := FALSE );
		IF NOT fbReceiveFrom.bBusy THEN
			IF NOT fbReceiveFrom.bError THEN
				IF fbReceiveFrom.nRecBytes > 0 THEN
					
					stReceivedFrom.stRemoteAddr.sAddr := fbReceiveFrom.sRemoteHost;
					stReceivedFrom.stRemoteAddr.nPort := fbReceiveFrom.nRemotePort;
					
					fbRx.AddTail( stPut := stReceivedFrom );
					IF NOT fbRx.bOk THEN(* Check for fifo overflow *)
						fbLog.Error( sMessage :='FB_FrameFifo(receiver)', nErrID := PLCPRJ_ERROR_RECFIFO_OVERFLOW );
					END_IF
				END_IF
				eStep := eUDP_STATE_IDLE;
			ELSE
				fbLog.Error( sMessage := 'FB_SocketUdpReceiveFrom()', nErrID := fbReceiveFrom.nErrID );
				IF fbReceiveFrom.nErrID = 16#80072746 THEN(* Connection is reset by remote side *)
					eStep := eUDP_STATE_IDLE;
				ELSE
					eStep := eUDP_STATE_ERROR;
				END_IF
			END_IF
		END_IF

	eUDP_STATE_CLOSE_START:
		fbLog.Message( sMessage := 'Closing connectionless (UDP) socket!', hSocket := fbCreate.hSocket );
		fbClose( bExecute := FALSE );
		fbClose( sSrvNetId := sSrvNetId, hSocket := fbCreate.hSocket, bExecute := TRUE );
		eStep := eUDP_STATE_CLOSE_WAIT;

	eUDP_STATE_CLOSE_WAIT:
		fbClose( bExecute := FALSE );
		IF NOT fbClose.bBusy THEN
			bCreated := FALSE;
			IF NOT fbClose.bError THEN
				eStep := eUDP_STATE_IDLE;
			ELSE
				fbLog.Error( sMessage := 'FB_SocketClose()', nErrID := fbClose.nErrID );
				eStep := eUDP_STATE_ERROR;
			END_IF
		END_IF

	eUDP_STATE_ERROR: (* Error step *)
		IF bCreated THEN
			eStep := eUDP_STATE_CLOSE_START;
		ELSE
			eStep := eUDP_STATE_IDLE;
		END_IF
END_CASE
*)

END_FUNCTION_BLOCK

// ---- POUs/Helper POUs/FB_FrameFifo.TcPOU
(* Tx/Rx (string data) fifo control function block *)
FUNCTION_BLOCK FB_FrameFifo
VAR_INPUT
	bLog		: BOOL := FALSE;(* TRUE => Enable log message output, FALSE => Disable *)
	sPrefix		: STRING := 'Unknown::';(* Log message description string (allows the identification of log message source) *)
	stPut		: ST_FrameFifoEntry;(* Frame entry to add (write) to the buffer *)
END_VAR
VAR_OUTPUT
	bOk			: BOOL;(* TRUE = New entry added or removed succesfully, FALSE = Fifo overflow or fifo empty *)
	stGet		: ST_FrameFifoEntry;(* Frame entry removed (read) from fifo *)
	nCount		: UDINT := 0;(* Number of fifo entries *)
END_VAR
VAR
	fbBuffer 	: FB_MemRingBuffer;(* Basic (lower level) string buffer control function block *)
	buffer		: ARRAY[0..PLCPRJ_BUFFER_SIZE] OF BYTE;(* Internal buffer memory *)
END_VAR

;

ACTION AddTail:
(* Adds new fifo entry *)
fbBuffer.A_AddTail( pBuffer:= ADR(buffer), cbBuffer:= SIZEOF(buffer),
					pWrite:= ADR( stPut ), cbWrite := SIZEOF( stPut ), 
					bOk=>bOk, nCount=>nCount );
IF bOk AND bLog THEN(* Log message *)
	ADSLOGSTR( ADSLOG_MSGTYPE_HINT OR ADSLOG_MSGTYPE_LOG, 
			CONCAT( CONCAT( sPrefix, SOCKETADDR_TO_STRING(stPut.stRemoteAddr) ), '>>"%s"' ),
			stPut.sMessage );
END_IF
END_ACTION

ACTION Clear:
(* Clears all fifo entries *)
stGet.sMessage := '';
stGet.stRemoteAddr.nPort := 0;
stGet.stRemoteAddr.sAddr := '';
fbBuffer.A_Reset( pBuffer := ADR( buffer ), cbBuffer := SIZEOF( buffer ), 
					bOk=>bOk, nCount=>nCount );
END_ACTION

ACTION RemoveHead:
(* Removes oldest fifo entry *)
IF nCount = 0 THEN
	stGet.sMessage := '';
	stGet.stRemoteAddr.nPort := 0;
	stGet.stRemoteAddr.sAddr := '';
	bOk := FALSE;
	RETURN;
END_IF

fbBuffer.A_RemoveHead( pBuffer:= ADR(buffer), cbBuffer:= SIZEOF(buffer),
						pRead := ADR( stGet ), cbRead := SIZEOF( stGet ),
						bOk=>bOk, nCount=>nCount );
END_ACTION

END_FUNCTION_BLOCK

// ---- POUs/Helper POUs/FB_LogFifo.TcPOU
(* Log/debug/error message fifo *)
FUNCTION_BLOCK FB_LogFifo
VAR_INPUT
	bLog		: BOOL 		:= FALSE;(* TRUE => Enable log message output, FALSE => Disable *)
	sPrefix		: STRING 	:= 'Unknown::';(* Log message description string (allows the identification of log message source) *)
	
	sMessage	: STRING 	:= '';(* String message to add (write) to the fifo *)
	nErrID		: UDINT 	:= 0;(* Error code to add (write) to the fifo *)
	hSocket		: T_HSOCKET;(* Socket connection handle *)
END_VAR
VAR_OUTPUT
	bOk			: BOOL;(* TRUE = New entry added or removed succesfully, FALSE = Fifo overflow or fifo empty *)
	sGet		: T_MaxString := '';(* String entry removed (read) from fifo *)
	nCount		: UDINT := 0;(* Number of fifo entries *)
END_VAR
VAR
	fbBuffer 	: FB_StringRingBuffer;(* Basic (lower level) string buffer control function block *)
	buffer		: ARRAY[0..PLCPRJ_BUFFER_SIZE] OF BYTE;(* Internal buffer memory *)
	sSource		: T_MaxString;	
	sPut		: T_MaxString;
END_VAR

;

ACTION Clear:
(* Clears all fifo entries *)
fbBuffer.A_Reset( 	pBuffer := ADR( buffer ), cbBuffer := SIZEOF( buffer ), 
					bOk=>bOk, nCount=>nCount, getValue=>sGet );
END_ACTION

ACTION Error:
(* Adds new fifo entry *)
IF nErrID = 0 THEN
	sSource := '::Error: 0x';
ELSIF ( nErrID AND 16#80000000) = 16#80000000 THEN
	IF nErrID = 16#80072746 THEN
		sSource := '::Win32 error (the connection is reset by remote side): 0x';
	ELSE
		sSource := '::Win32 error: 0x';
	END_IF
ELSIF (nErrID AND 16#00008100) = 16#00008100 THEN
	CASE nErrID OF
		PLCPRJ_ERROR_SENDFIFO_OVERFLOW:
			sSource := '::PLC sample project send fifo overflow error: 0x';
		PLCPRJ_ERROR_RECFIFO_OVERFLOW:
			sSource := '::PLC sample project receive fifo overflow error: 0x';
	ELSE
		sSource := '::Other PLC sample project error: 0x';
	END_CASE
ELSIF (nErrID AND 16#00008000) = 16#00008000 THEN
	sSource := '::Internal TCP/IP Connection Server error: 0x';
ELSE
	sSource := '::TwinCAT System error: 0x';
END_IF

sPut := CONCAT( CONCAT( CONCAT( sPrefix, sMessage ), sSource ), DWORD_TO_HEXSTR( nErrID AND 16#FFFF, 0, FALSE ) ); 

fbBuffer.A_AddTail( pBuffer:= ADR(buffer), cbBuffer:= SIZEOF(buffer),
					putValue:= sPut, bOk=>bOk, nCount=>nCount );
IF bOk THEN
	IF bLog THEN(* Log error message *)
		ADSLOGSTR( ADSLOG_MSGTYPE_ERROR OR ADSLOG_MSGTYPE_LOG, '%s', sPut );	
	END_IF
END_IF
END_ACTION

ACTION Message:
(* Adds new fifo entry *)
sPut := CONCAT( CONCAT( sPrefix, sMessage ), CONCAT( '::', SOCKETADDR_TO_STRING(hSocket.localAddr) ) );
fbBuffer.A_AddTail( pBuffer:= ADR(buffer), cbBuffer:= SIZEOF(buffer),
					putValue:= sPut, bOk=>bOk, nCount=>nCount );
IF bOk THEN
	IF bLog THEN(* Log information message *)
		ADSLOGSTR( ADSLOG_MSGTYPE_HINT OR ADSLOG_MSGTYPE_LOG, '%s', sPut );	
	END_IF
END_IF
END_ACTION

ACTION Remove:
(* Removes oldest fifo entry *)
IF nCount = 0 THEN
	sGet := '';
	bOk := FALSE;
	RETURN;
END_IF

fbBuffer.A_RemoveHead( pBuffer:= ADR(buffer), cbBuffer:= SIZEOF(buffer),
						getValue=>sGet, bOk=>bOk, nCount=>nCount );
END_ACTION

END_FUNCTION_BLOCK

// ---- POUs/Control_LIbs/FT_DERIV_1.TcPOU
FUNCTION_BLOCK FT_DERIV_1
VAR_INPUT
	in : REAL;
	K : REAL := 1.0;
	run : BOOL := TRUE;
END_VAR
VAR_OUTPUT
	out : REAL;
END_VAR
VAR
	old: REAL;
	tx: DWORD;
	last: DWORD;
	init: BOOL;
	tc: REAL;
END_VAR


(*
version 1.5	11. mar. 2009
programmer 	hugo
tested by		oscat

FT_deriv calculates the derivate over the signal "in" with Faktor "K".
a run input enables or stops the calculation, if left unconnected its true and therfore the calculation is executed.
if K is not specified the default is 1.

*)

(* read system time *)
tx := T_PLC_US();
tc := DWORD_TO_REAL(tx - last);
last := tx;

(* init on first startup *)
IF NOT init THEN
	init := TRUE;
	old := in;
ELSIF run AND tc > 0.0 THEN
	out := (in - old) / tc * 1000000.0 * K;
	old := in;
ELSE
	out := 0.0;
END_IF;



(*
hm 3.1.2007			rev 1.1
	added init code for startup
	set the default for K to 1

hm	15. sep 2007	rev 1.2
	replaced Time() with T_PLC_US for compatibility and performance reasons
	increased accuracy and work in microseconds internally

hm 29 oct 2007	rev 1.3
	prohibit calculation when tx - last = 0 to avoid division by 0 and increase accuracy on fast systems

hm	6. nov. 2008	rev 1.4
	improved performance

hm	11. mar. 2009	rev 1.5
	inproved code
*)

END_FUNCTION_BLOCK

// ---- POUs/Control_LIbs/FT_INT.TcPOU
FUNCTION_BLOCK FT_INT
VAR_INPUT
	IN : REAL;
	K : REAL := 1;
	RUN : BOOL := TRUE;
	RST : BOOL;
	OUT_MIN : REAL := -1E37;
	OUT_MAX : REAL := 1E37;
END_VAR
VAR_OUTPUT
	OUT : REAL;
	LIM : BOOL;
END_VAR
VAR
	INTeg : INTEGRATE;
END_VAR


(*
version 2.2	10. mar. 2009
programmer 	hugo
tested by		oscat

FT_int is an integrator with input IN and factor K.
integration is only done while run = true, if run is false integration is stopped and the out remains at the last value.
if run is left unconnected, run is considered true by the function block.
the output ET will display the total integration time from last reset.
the out_min and out_max values can be set to ,imit the output value range. 
the default for K is 1.

 
*)

IF rst THEN
	out := 0.0;
ELSE
	integ(X := IN, E := RUN, K := K, Y := out);
END_IF;

(* limit the outputs *)
IF out >= OUT_MAX THEN
	out := out_max;
	LIM := TRUE;
ELSIF out <= out_min THEN
	out := out_min;
	lim := TRUE;
ELSE
	lim := FALSE;
END_IF;


(*
hm 13.12.2006	rev 1.1
	changed to "trapezregel" which increases accuracy
	before out := out + in * time new: out := out + (in + in_last) / 2 * time

hm 15.1.2007		rev 1.2
	added default for k to be 1.

hm	15.9.2007		rev 1.3
	replaced time() with T_PLC_US for compatibility and performance reason
	increased internal accuracy to microseconds

hm 29. oct 2007		rev 1.4
	changed code so int will not be called is time difference is 0 to increase accuracy on systems
	with cycle times below 1ms

hm	2. dec 2007	 	rev 1.5
	changed code for better performance

hm	5. jan 2008		rev 1.6
	further improvements in performance

hm	8. feb 2008		rev 1.7
	deleted limits +/- 1000 now limit is the range of real
	added variables out1 and out2 to extend the resolution
	corrected an error with elapsed time
	deleted unusfull output ET

hm	13. mar 2008	rev 1.8
	changed preset value out_min to -1e37.
	stop integrator at the limits.

hm	16. mar 2008	rev 1.9
	added type conversion to avoid warning under codesys 3.0

hm	2. jun. 2008	rev 2.0
	rewritten with clear code
	limits can now be set without run

hm	3. nov. 2008	rev 2.1
	optimized code using INTEGRATE and LIMX

hm	10. mar. 2009	rev 2.2
	removed nested comments
*)

END_FUNCTION_BLOCK

// ---- POUs/Control_LIbs/INTEGRATE.TcPOU
FUNCTION_BLOCK INTEGRATE
VAR_INPUT
	E : BOOL := TRUE;
	X : REAL;
	K : REAL := 1.0;
END_VAR
VAR_IN_OUT
	Y : REAL;
END_VAR
VAR
	X_last : REAL;
	init: BOOL;
	last: DWORD;
	tx: DWORD;
END_VAR


(*
version 1.0	3. nov. 2008
programmer 	hugo
tested by	oscat

integrate is a plain integrator with I/O for out.

 
*)

(*read system time *)
tx := T_PLC_MS();

IF NOT init THEN
	init := TRUE;
	X_last := X;
ELSIF E THEN
	Y := (X + X_LAST) * 0.5E-3 * DWORD_TO_REAL(tx-last) * K + Y;
	X_last := X;
END_IF;
last := tx;



(*
hm 3. nov. 2008	rev 1.0
original version
	
*)

END_FUNCTION_BLOCK

// ---- POUs/Control_LIbs/FT_PID.TcPOU
FUNCTION_BLOCK FT_PID
VAR_INPUT
	IN : REAL;
	KP : REAL := 1.0;
	TN : REAL := 1.0;
	TV : REAL := 1.0;
	ILIM_L : REAL := -1.0E38;
	ILIM_H : REAL := 1.0E38;
	IEN : BOOL := TRUE;
	RST : BOOL;
END_VAR
VAR_OUTPUT
	Y : REAL;
	LIM : BOOL;
END_VAR
VAR
	integ : FT_INT;
	diff : FT_DERIV;
END_VAR

(*
version 2.1	11. mar. 2009
programmer 	hugo
tested by		tobias

FT_PI is a PI controller.
The PID controller works according to the fomula Y = IN *(KP+ KI * INTEG(e) ).
a rst will reset the integrator to 0
ilim_h and iLim_l set the possible output range of the internal integrator.
the output flags lim will signal that the output limits are active.

default values for KP = 1, KI = 1, ILIM_L = -1E37, iLIM_H = +1E38.
*)

(* run integrator only if TN > 0 *)
IF TN > 0.0 THEN
	integ(IN := IN, K := 1.0 / TN, RUN := IEN, RST := RST, OUT_MIN := ILIM_L, OUT_MAX := ILIM_H);
ELSE
	integ(RST := FALSE);
END_IF;

(* run differentiator *)
diff(IN := IN, K := TV);

(* combine both values *)
Y := KP * (integ.Out + diff.out + IN);

(* check if integrator has reached its limits and set overflow *)
LIM := integ.LIM;



(* revision history
hm 3. jun. 2008 	rev 2.0
	original version

hm	11. mar. 2009	rev 2.1
	real constants updated to new systax using dot

*)

END_FUNCTION_BLOCK

// ---- GlobalTextList.TcGTLO
TEXTLIST GlobalTextList
  3111 = ' Output PWM (%)'
  81 = '% s'
  243 = '%2.1 '
  184 = '%2.1f %'
  220 = '%2.1f (mbar)'
  2367 = '%2.1f (s)'
  188 = '%2.1f KI (%)'
  862 = '%2.1f KP '
  187 = '%2.1f KP (%)'
  2090 = '%2.1f Tn '
  264 = '%2.1f Tn (%)'
  124 = '%2.1f Value Comp PT100'
  245 = '%2.2f'
  1292 = '%2.2f '
  36 = '%2u'
  32 = '%2u '
  185 = '%2u %'
  1617 = '%2u (s)'
  2765 = '%2u 0-100%'
  2392 = '%2u 0-1400%'
  518 = '%2u 0-14001/min'
  91 = '%3.2f'
  103 = '%3.2f  '
  152 = '%3.2f  (mbar)'
  50 = '%3.2f  (°C)'
  217 = '%3.2f  Heizband2'
  218 = '%3.2f  Heizband3'
  314 = '%3.2f  Ps_202'
  3063 = '%3.2f  Ps_203'
  141 = '%3.2f  SEO2 1.51'
  122 = '%3.2f  SEP1.11'
  1831 = '%3.2f  SEP1.12'
  631 = '%3.2f  SEP1.13'
  119 = '%3.2f  SEP2.11'
  121 = '%3.2f  SEP2.12'
  248 = '%3.2f  SEP2.13'
  2143 = '%3.2f  SEP2.14'
  90 = '%3.2f  SET2.8'
  227 = '%3.2f  SET3.8'
  142 = '%3.2f  SEW 2.31'
  219 = '%3.2f  T.Mittel'
  2227 = '%3.2f  VolFracAir1'
  1505 = '%3.2f  VolFracAir1202'
  497 = '%3.2f  VolFracAir202'
  1959 = '%3.2f  VolFracAir203'
  2102 = '%3.2f  volFracAirO2'
  205 = '%3.2f (ms)'
  149 = '%3.2f Comp.L1'
  150 = '%3.2f Comp.L2'
  151 = '%3.2f Comp.L3'
  99 = '%3.2f Heatreg 2'
  2982 = '%3.2f Heatreg compressor'
  100 = '%3.2f Heatreg1'
  1670 = '%3.2f Heatreg1-4'
  128 = '%3.2f Heatreg2'
  101 = '%3.2f Heatreg3'
  157 = '%3.2f Heatreg4'
  158 = '%3.2f Heatreg5'
  899 = '%3.2f Heatreg5-8'
  159 = '%3.2f Heatreg6'
  160 = '%3.2f Heatreg7'
  161 = '%3.2f Heatreg8'
  146 = '%3.2f Main L1'
  147 = '%3.2f Main L2'
  148 = '%3.2f Main L3'
  444 = '%3.2f PS202'
  109 = '%3.2f SET 1.01'
  110 = '%3.2f SET 1.02 '
  2829 = '%3.2f SET 1.03'
  111 = '%3.2f SET 1.03 '
  112 = '%3.2f SET 1.04 '
  113 = '%3.2f SET 1.05'
  114 = '%3.2f SET 1.06'
  115 = '%3.2f SET 1.07'
  116 = '%3.2f SET 1.08'
  117 = '%3.2f SET 1.09'
  173 = '%3.2f SET 1.81 '
  174 = '%3.2f SET 1.82'
  175 = '%3.2f SET 1.83'
  176 = '%3.2f SET 1.91'
  177 = '%3.2f SET 1.92'
  178 = '%3.2f SET 1.93'
  162 = '%3.2f SET 2.01'
  163 = '%3.2f SET 2.02 '
  164 = '%3.2f SET 2.03 '
  2577 = '%3.2f SET 203 '
  165 = '%3.2f SET 3.01 '
  166 = '%3.2f SET 3.02'
  167 = '%3.2f SET 3.03'
  1934 = '%3.2f SET 3.51'
  168 = '%3.2f SET 3.71'
  169 = '%3.2f SET 3.72'
  170 = '%3.2f SET 3.73'
  171 = '%3.2f SET 3.74'
  2317 = '%3.2f SET 3.75'
  738 = '%3.2f SET 3.76'
  553 = '%3.2f SET 3.77'
  2540 = '%3.2f SET 3.78'
  179 = '%3.2f SET 3.81'
  180 = '%3.2f SET 3.82'
  181 = '%3.2f SET 3.83'
  182 = '%3.2f SET 3.84'
  2060 = '%3.2f SET 3.85'
  607 = '%3.2f SET 3.86'
  2031 = '%3.2f SET 3.87'
  1483 = '%3.2f SET 3.88'
  172 = '%3.2f SET 4.01'
  140 = '%3.2f SET Ambiente'
  2324 = '%3.2f STG L1'
  569 = '%3.2f STG L2'
  1438 = '%3.2f STG L3'
  236 = '%3.2f Tauch-HZ. L1'
  235 = '%3.2f Tauch-HZ. L2'
  234 = '%3.2f Tauch-HZ. L3'
  125 = '%3.2f UD  L1'
  126 = '%3.2f UD  L2'
  127 = '%3.2f UD  L3'
  130 = '%3u Temp. Heatmatt1 '
  139 = '%3u Temp. Heatmatt10 '
  131 = '%3u Temp. Heatmatt2 '
  132 = '%3u Temp. Heatmatt3 '
  133 = '%3u Temp. Heatmatt4 '
  134 = '%3u Temp. Heatmatt5 '
  135 = '%3u Temp. Heatmatt6 '
  136 = '%3u Temp. Heatmatt7 '
  137 = '%3u Temp. Heatmatt8'
  138 = '%3u Temp. Heatmatt9 '
  24 = '%s'
  191 = 'Activate'
  20 = 'Advanced\nControl'
  186 = 'Ausgabe Stellwert'
  17 = 'Auto'
  87 = 'Auto active'
  92 = 'Auto-Output'
  1577 = 'Back'
  1699 = 'back'
  28 = 'Check Comp\nTemperature!'
  257 = 'Close HMI'
  27 = 'Continue\nStartup'
  68 = 'Current Total [A]'
  728 = 'Dampf-'
  2667 = 'Dampf-\nGenerator'
  86 = 'Default=Auto active'
  216 = 'DO1'
  230 = 'DO2'
  233 = 'DO3'
  231 = 'DO4'
  120 = 'Druck (mBar):'
  25 = 'Durchmesser in mm eingeben'
  98 = 'Duty Cycle'
  69 = 'Electrical Power [kW]'
  2986 = 'Error O2'
  344 = 'forward'
  991 = 'Frequence (HZ) \nmax. 0.02=50s'
  2936 = 'Frequence (HZ) max. 0.02'
  2404 = 'Frequence (HZ) max. 0.02=50s'
  40 = 'FU OK'
  38 = 'FU ON'
  13 = 'Group1'
  12 = 'Group2'
  11 = 'Group3'
  97 = 'Hauptschütz'
  2425 = 'Heat \nController'
  250 = 'Heat Controller'
  2040 = 'Heat Output PWM (%)'
  2689 = 'Heat Output Set (%)'
  155 = 'Heatregister'
  1816 = 'Heizband'
  226 = 'Heizeinschraubkörper:'
  74 = 'Heizelemente ON/OFF'
  10 = 'Heizmatten'
  73 = 'Heizmatten ON/OFF'
  143 = 'Heizmatten:'
  2987 = 'Heizregister 1'
  244 = 'Heizregister 2'
  215 = 'Heizregister Kompressor'
  89 = 'Heizregister:'
  85 = 'Heizreglerbetrieb:'
  966 = 'Heizungen'
  3471 = 'Horizontalband oben'
  3473 = 'Horizontalband unten'
  43 = 'Hysterese hoch (°C)'
  42 = 'Hysterese tief (°C)'
  2600 = 'I-Anteil'
  210 = 'In Progress'
  223 = 'Integralwert'
  2313 = 'Istwert'
  225 = 'Istwert Vordruck Scrolli'
  720 = 'K-Anteil'
  154 = 'Kompressor'
  153 = 'Kompressoreinlass'
  228 = 'L1:'
  229 = 'L2:'
  232 = 'L3:'
  527 = 'Lampe'
  2114 = 'Layout'
  752 = 'Main'
  14 = 'Main ON'
  1499 = 'Main ON/OFF'
  94 = 'Main-Output'
  129 = 'Main: in (A)'
  19 = 'Manu'
  93 = 'Manu-Output'
  34 = 'MANUEL BETRIEB'
  955 = 'MANUELBETRIEB'
  0 = 'Mat1'
  9 = 'Mat10'
  2 = 'Mat2'
  4 = 'Mat3'
  6 = 'Mat4'
  8 = 'Mat5'
  1 = 'Mat6'
  3 = 'Mat7'
  5 = 'Mat8'
  7 = 'Mat9'
  2780 = 'Mindest einschaltzeit puls (S)'
  207 = 'Next Step'
  2895 = 'Nicht aussschalten unter 20%'
  345 = 'O2'
  1277 = 'O2 Heat ON'
  29 = 'OK for \nOperation'
  88 = 'ON/OFF'
  23 = 'ON1'
  22 = 'ON2'
  21 = 'ON3'
  2677 = 'P-Anteil'
  1085 = 'Periodendauer PWM (S)'
  368 = 'PID'
  71 = 'Press. Umg'
  224 = 'Proportionalwert'
  1185 = 'PWM Cycle (%) max.100'
  33 = 'PWM Output 0-100%'
  2990 = 'Recalibrate P-Sensors'
  1869 = 'Recalibrate TC-Sensors'
  96 = 'Ref. Temp'
  903 = 'Regelparameter Heizreister oben'
  183 = 'Regelparameter Kompressor Klauenkolben'
  193 = 'Regelparameter Kompressor Scrolli'
  192 = 'Regelparameter Nadelventil'
  61 = 'Rel. P OUT'
  62 = 'Rel. P TM'
  54 = 'Rel. P WT'
  18 = 'Reset'
  15 = 'Reset '
  2126 = 'Reset Calib P-Sensors'
  3182 = 'Reset Calib TC-Sensors'
  213 = 'Reset Seq.'
  67 = 'RPM Des. Venti [%]'
  65 = 'RPM Kompressor [%]'
  238 = 'S'
  209 = 'Schrittnummer:'
  37 = 'Schütz'
  1696 = 'Schütz1'
  2308 = 'Schütz2'
  59 = 'SE-P2.2'
  56 = 'SE-P2.5'
  64 = 'SE-P3.11'
  57 = 'SE-P3.3'
  76 = 'SE-P3.32'
  63 = 'SE-P6.2'
  60 = 'SE-T2.3'
  78 = 'SE-T2.51'
  80 = 'SE-T2.52'
  55 = 'SE-T2.6'
  53 = 'SE-T2.8'
  70 = 'SE-T3.31'
  77 = 'SE-T3.33'
  58 = 'SE-T3.4'
  66 = 'SE-T3.51'
  79 = 'SE-T3.52'
  869 = 'Send Trigger'
  241 = 'Sensors'
  212 = 'Sequence End'
  2084 = 'Service'
  2578 = 'Service2'
  95 = 'Setpoint'
  242 = 'Show'
  123 = 'Sicherheitstemps:'
  239 = 'Sollwert'
  190 = 'Sollwert Druck Dampfkammer'
  49 = 'Sollwert Horizontalband'
  1009 = 'Sollwert Horizontalband  '
  2585 = 'Sollwert Horizontalband oben'
  39 = 'Sollwert Kompressor'
  3156 = 'Sollwert min: 0.41/min bis 1.6 1/min'
  2399 = 'Sollwert min:0.081/min bis 0.48 1/min'
  246 = 'Sollwert min:0.41/min bis 1.6 1/min'
  222 = 'Sollwert Primär Kompressor'
  52 = 'Sollwert Steigförderer'
  2074 = 'Sollwert Temp Heatreg oben'
  370 = 'Sollwert Umdampfventi'
  35 = 'Sollwert Umdampfventilator'
  221 = 'Sollwert Vordruck Scrolli'
  2132 = 'Sollwert xy'
  26 = 'Start\nAutostart'
  208 = 'Start Again'
  211 = 'Start Point'
  30 = 'Startup\nfinished'
  31 = 'Startup Active'
  1383 = 'Steamfan OK'
  657 = 'Steamfan OK\nfor heating'
  247 = 'Steamfan OK\nfor heating\nmin 25% volume'
  1676 = 'Steamfan OK\nfot heating'
  249 = 'Steigförderer'
  189 = 'Stellwert Kompressor Manu'
  214 = 'Step back'
  102 = 'Stromverbrauch: in (A)'
  2996 = 'switch'
  2967 = 'switch\nInput'
  1132 = 'switch\nPWM'
  16 = 'Switch OFF'
  627 = 'Switch OFF\t'
  556 = 'T 1.03 Heizregister'
  2413 = 'T 1.04 Heizregister'
  418 = 'T 1.05 Regeltemperatur'
  1616 = 'T 1.06 Regeltemperatur'
  2645 = 'T 4.01 Heizband'
  1043 = 'T.Monitor '
  105 = 'T.Monitor 1 SE-T 1.03'
  107 = 'T.Monitor 1 SE-T 1.04'
  106 = 'T.Monitor 2 SE-T 1.05'
  108 = 'T.Monitor 2 SE-T 1.06'
  2391 = 'T.Monitor Mean Values'
  2101 = 'T.Monitor Mean Values  '
  2587 = 'T.Monitor xy'
  41 = 'Temp\nError'
  145 = 'Temp\nError comp.'
  144 = 'Temp\nError SteamFan'
  1489 = 'Temp. \nKompressor \nGehause'
  237 = 'Temp. \nKompressor Gehause'
  51 = 'Temp. Kompressor Gehause'
  72 = 'Temp. Umg'
  118 = 'Temperaturen (°C):'
  104 = 'Tempimit switch OFF (°C)\ngroup TOP'
  2474 = 'Tempimit switch OFF (°C)\nHeizband'
  1589 = 'Testseite'
  75 = 'TM'
  2371 = 'UDP-Kommunikation'
  156 = 'Umdampfventi'
  1817 = 'Umrechnungen'
  240 = 'V Main'
  203 = 'V-Dichtring\nAuslass'
  202 = 'V-Dichtring\nEinlass'
  47 = 'V1'
  44 = 'V2'
  45 = 'V3'
  46 = 'V4'
  48 = 'V5'
  1447 = 'V6'
  196 = 'Vacuum1'
  195 = 'Vacuum2'
  1501 = 'VE-K 2.71\n\n\nVE-K 2.72\n\n\nVE-K 2.73'
  829 = 'VE-K 2.71\n\nVE-K 2.72\n\nVE-K 2.73'
  84 = 'VE-K 2.71\n\nVE-K 2.73'
  1371 = 'VE-K 2.71\n\nVE-K 3.71\n\nVE-K 3.72'
  82 = 'VE-K2.71'
  511 = 'VE-K2.72'
  83 = 'VE-K2.73'
  194 = 'VE-K3.05'
  197 = 'VE-K3.06'
  198 = 'VE-K3.13'
  199 = 'VE-K3.19'
  200 = 'VE-K3.20'
  201 = 'VE-K3.21'
  204 = 'VE-K3.22'
  1148 = 'VE-K3.71'
  964 = 'VE-K3.72'
  3206 = 'Wasserverdampfer'
  206 = 'Zykluszeit Reglerausgnag (ms)'
END_TEXTLIST

// ---- Visualizations/PID.TcVIS
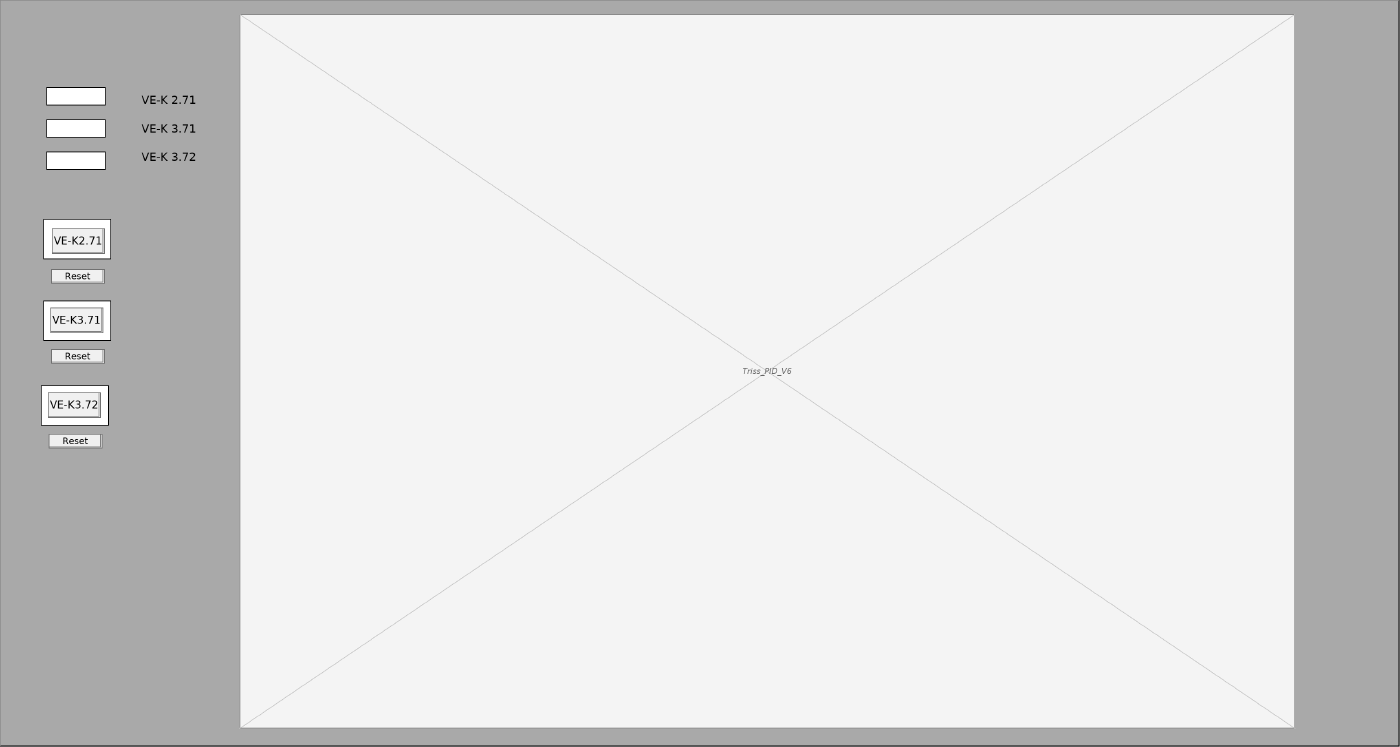
VISUALIZATION PID  // 1782x952, background image 
    Rectangle (0,950 1780x2)
    Rectangle (1780,0 2x950)
    Rectangle (55,279 86x51), colour toggle: GVL.V_Dampf_nach_Komp
    Button (66,291 67x32), "VE-K2.71"
        tap GVL.V_Dampf_nach_Komp_manu
    Button (65,343 68x18), "Reset"
        tap GVL.V_Dampf_nach_Komp_Reset
    Rectangle (55,383 86x51), colour toggle: V_Entlueftung_1
    Button (64,392 67x32), "VE-K3.71"
        tap V_Entlueftung_1_manu
    Button (65,445 68x18), "Reset"
        tap V_Entlueftung_1_Reset
    Rectangle (59,111 75x23), colour toggle: GVL.V_Dampf_nach_Komp_negiert
    Rectangle (59,152 75x23), colour toggle: V_Entlueftung_1_negiert
    Rectangle (143,86 144x156), "VE-K 2.71 VE-K 3.71 VE-K 3.72"
    Rectangle (52,491 86x51), colour toggle: V_Entlueftung_2
    Button (61,500 67x32), "VE-K3.72"
        tap V_Entlueftung_2_manu
    Button (62,553 68x18), "Reset"
        tap GVL.V_Entlueftung_2_Reset
    Rectangle (59,193 75x23), colour toggle: V_Entlueftung_2_negiert
    Image (305,18 1343x910), image: Triss_PID_V6
END_VISUALIZATION

// ---- Visualizations/Main.TcVIS
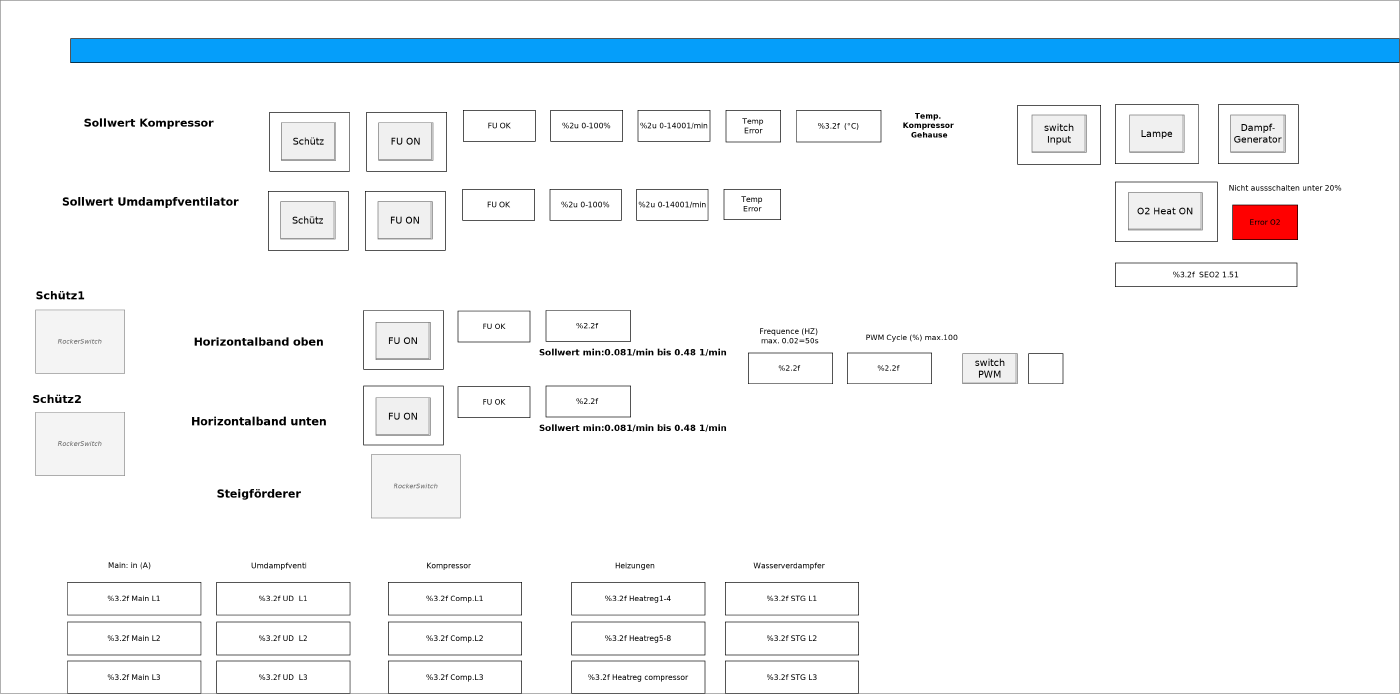
VISUALIZATION Main  // 2147x1065, background image backround
    Rectangle (1560,161 128x91), colour toggle: switch_Setpoint_Value
    Rectangle (108,59 2039x37)
    Rectangle (844,169 111x48), "%2u 0-100%", tooltip "Durchmesser in mm eingeben", text variable: GVL.Setpoint_Compressor_Visu
        OnMouseDown: write the text variable via VisuDialogs.Numpad, min 0, max 100
    Rectangle (837,592 130x48), "%2.2f", text variable: Setpoint_Belts_Visu_bottom_1_min
        OnMouseDown: write the text variable via VisuDialogs.Numpad, min 0.0, max 0.48
    Rectangle (1113,169 84x49), "Temp Error", colour toggle: GVL.Compressor_PT100_error
    Rectangle (843,290 110x48), "%2u 0-100%", tooltip "Durchmesser in mm eingeben", text variable: GVL.Setpoint_SteamFan_Visu
        OnMouseDown: write the text variable via VisuDialogs.Numpad, min 0, max 100
    Rectangle (1110,290 87x47), "Temp Error"
    Rectangle (1221,169 130x49), "%3.2f (°C)", tooltip "Durchmesser in mm eingeben", text variable: GVL.T_Ueberwachung_scroll_comp
    Rectangle (1339,161 173x63), "Temp. Kompressor Gehause"
    Textfield (84,172 288x33), "Sollwert Kompressor"
    Textfield (84,293 293x33), "Sollwert Umdampfventilator"
    Textfield (253,630 288x33), "Horizontalband unten"
    Textfield (253,741 288x33), "Steigförderer"
    Rectangle (411,293 123x91), colour toggle: GVL.SteamFAN_Switch_ON_manu
    Button (430,309 84x58), "Schütz", pressed state: GVL.SteamFAN_Switch_ON_manu
        toggle GVL.SteamFAN_Switch_ON_manu
    Rectangle (413,172 123x91), colour toggle: GVL.Compressor_Switch_ON_Manu
    Button (431,188 84x58), "Schütz", pressed state: GVL.Compressor_Switch_ON_Manu
        toggle GVL.Compressor_Switch_ON_Manu
    Rectangle (562,172 123x91), colour toggle: GVL.Compressor_ON_Manu
    Button (580,188 84x58), "FU ON", pressed state: GVL.Compressor_ON_Manu
        toggle GVL.Compressor_ON_Manu
    Rectangle (710,169 111x48), "FU OK", colour toggle: GVL.Compressor_OK
    Rectangle (709,290 111x48), "FU OK", colour toggle: GVL.SteamFan_OK
    Rectangle (557,592 123x91), colour toggle: GVL.Belts_ON_bottom_Manu
    Button (576,610 84x58), "FU ON", pressed state: GVL.Belts_ON_bottom_Manu
        toggle GVL.Belts_ON_bottom_Manu
    Rectangle (702,593 111x48), "FU OK", colour toggle: GVL.Belts_bottom_OK
    Rectangle (560,293 123x91), colour toggle: GVL.SteamFan_ON_manu
    Button (579,309 84x58), "FU ON"
        toggle GVL.SteamFan_ON_manu
    Rectangle (332,893 205x51), "%3.2f UD L1", tooltip "Durchmesser in mm eingeben", text variable: Current_OUT_Fan_L1
    Rectangle (332,954 205x51), "%3.2f UD L2", tooltip "Durchmesser in mm eingeben", text variable: Current_OUT_Fan_L2
    Rectangle (332,1014 205x51), "%3.2f UD L3", tooltip "Durchmesser in mm eingeben", text variable: Current_OUT_Fan_L3
    Rectangle (876,893 205x51), "%3.2f Heatreg1-4", tooltip "Durchmesser in mm eingeben", text variable: Current_OUT_Heatreg_1_TO_4
    Rectangle (876,954 205x51), "%3.2f Heatreg5-8", tooltip "Durchmesser in mm eingeben", text variable: Current_OUT_Heatreg_5_TO_8
    Rectangle (876,1014 205x51), "%3.2f Heatreg compressor", tooltip "Durchmesser in mm eingeben", text variable: Current_OUT_Heatreg_Compressor
    Rectangle (123,849 151x37), "Main: in (A)"
    Rectangle (103,893 205x51), "%3.2f Main L1", tooltip "Durchmesser in mm eingeben", text variable: GVL.Current_OUT_Complete_L1
    Rectangle (103,954 205x51), "%3.2f Main L2", tooltip "Durchmesser in mm eingeben", text variable: GVL.Current_OUT_Complete_L2
    Rectangle (103,1014 205x51), "%3.2f Main L3", tooltip "Durchmesser in mm eingeben", text variable: GVL.Current_OUT_Complete_L3
    Rectangle (595,893 205x51), "%3.2f Comp.L1", tooltip "Durchmesser in mm eingeben", text variable: GVL.Current_OUT_Compressor_L1
    Rectangle (595,954 205x51), "%3.2f Comp.L2", tooltip "Durchmesser in mm eingeben", text variable: GVL.Current_OUT_Compressor_L2
    Rectangle (595,1014 205x51), "%3.2f Comp.L3", tooltip "Durchmesser in mm eingeben", text variable: GVL.Current_OUT_Compressor_L3
    Rectangle (582,857 212x22), "Kompressor"
    Rectangle (849,857 250x22), "Heizungen"
    Rectangle (322,857 212x22), "Umdampfventi"
    Rectangle (1112,893 205x51), "%3.2f STG L1", tooltip "Durchmesser in mm eingeben", text variable: Current_OUT_SteamGen1
    Rectangle (1112,954 205x51), "%3.2f STG L2", tooltip "Durchmesser in mm eingeben", text variable: Current_OUT_SteamGen2
    Rectangle (1112,1014 205x51), "%3.2f STG L3", tooltip "Durchmesser in mm eingeben", text variable: Current_OUT_SteamGen3
    Rectangle (1085,857 250x22), "Wasserverdampfer"
    Rectangle (1710,160 128x91), colour toggle: MAIN_ON_Switch_Light_visu
    Button (1732,176 84x58), "Lampe", pressed state: GVL.Belts_TOP_Switch_ON_Manu, input disabled if: GVL.Control_Manu_active=False
        toggle MAIN_ON_Switch_Light_visu
    Rectangle (1868,160 123x91), colour toggle: MAIN_ON_STEAM_GEN
    Button (1887,176 84x58), "Dampf- Generator", pressed state: GVL.Belts_TOP_Switch_ON_Manu, input disabled if: GVL.Control_Manu_active=FALSE
        toggle MAIN_ON_STEAM_GEN
    Textfield (805,642 331x30), "Sollwert min:0.081/min bis 0.48 1/min"
    Rectangle (1710,403 279x37), "%3.2f SEO2 1.51", tooltip "Durchmesser in mm eingeben", text variable: GVL.O2_Visu
    Rectangle (1710,279 157x92), colour toggle: O2_Sensor_Start
    Button (1730,295 114x58), "O2 Heat ON", pressed state: GVL.Belts_TOP_Switch_ON_Manu, input disabled if: DO_not_turn_off_Heating_O2_Sensor
        toggle O2_Sensor_Start
    Rectangle (1890,314 100x54), "Error O2", colour toggle: O2_Sensor_Error
    Rectangle (1862,270 218x37), "Nicht aussschalten unter 20%"
    Rectangle (978,169 111x48), "%2u 0-14001/min", tooltip "Durchmesser in mm eingeben", text variable: Setpoint_1_MIN_Compressor_IN
        OnMouseDown: write the text variable via VisuDialogs.Numpad, min 0, max 100
    Rectangle (976,290 110x48), "%2u 0-14001/min", tooltip "Durchmesser in mm eingeben", text variable: GVL.Setpoint_SteamFan_Visu
        OnMouseDown: write the text variable via VisuDialogs.Numpad, min 0, max 100
    Button (1582,176 84x58), "switch Input", pressed state: GVL.Belts_TOP_Switch_ON_Manu
        toggle switch_Setpoint_Value p2164770859=TRUE
    Rectangle (837,476 130x48), "%2.2f", text variable: Setpoint_Belts_Visu_TOP_1_min
        OnMouseDown: write the text variable via VisuDialogs.Numpad, min 0.0, max 0.48
    Textfield (253,508 288x33), "Horizontalband oben"
    Rectangle (557,476 123x91), colour toggle: GVL.Belts_ON_TOP_Manu
    Button (576,494 84x58), "FU ON", pressed state: GVL.Belts_ON_TOP_Manu
        toggle GVL.Belts_ON_TOP_Manu
    Rectangle (702,477 111x48), "FU OK", colour toggle: GVL.Belts_OK_TOP
    Textfield (805,526 331x30), "Sollwert min:0.081/min bis 0.48 1/min"
    Rectangle (1147,541 130x48), "%2.2f", text variable: Base_Frequence_Main_Belt
        OnMouseDown: write the text variable via VisuDialogs.Numpad, min 0, max 10
    Rectangle (1299,541 130x48), "%2.2f", text variable: Main_Belt_PWMDutyCycle_VISU
        OnMouseDown: write the text variable via VisuDialogs.Numpad, min 20, max 100
    Rectangle (1143,496 137x40), "Frequence (HZ) max. 0.02=50s"
    Rectangle (1304,507 189x22), "PWM Cycle (%) max.100"
    Rectangle (1577,542 53x47), colour toggle: Switch_ON_Main_Belt_PWM
    Button (1476,542 84x47), "switch PWM", pressed state: GVL.Belts_TOP_Switch_ON_Manu
        toggle Switch_ON_Main_Belt_PWM p2164770859=TRUE
    RockerSwitch (54,475 137x98), variable: Circuit_1_ON, behaviour: TOGGLE, style: Switch-RockerSwitch-Gray
    RockerSwitch (54,632 137x98), variable: Circuit_2_ON, behaviour: TOGGLE, style: Switch-RockerSwitch-Gray
    RockerSwitch (569,697 137x98), variable: GVL.M_Belt_Feeder_ON_Manu, behaviour: TOGGLE, style: Switch-RockerSwitch-Gray
    Textfield (29,437 127x33), "Schütz1"
    Textfield (24,596 127x33), "Schütz2"
END_VISUALIZATION

// ---- Visualizations/PID_alt.TcVIS
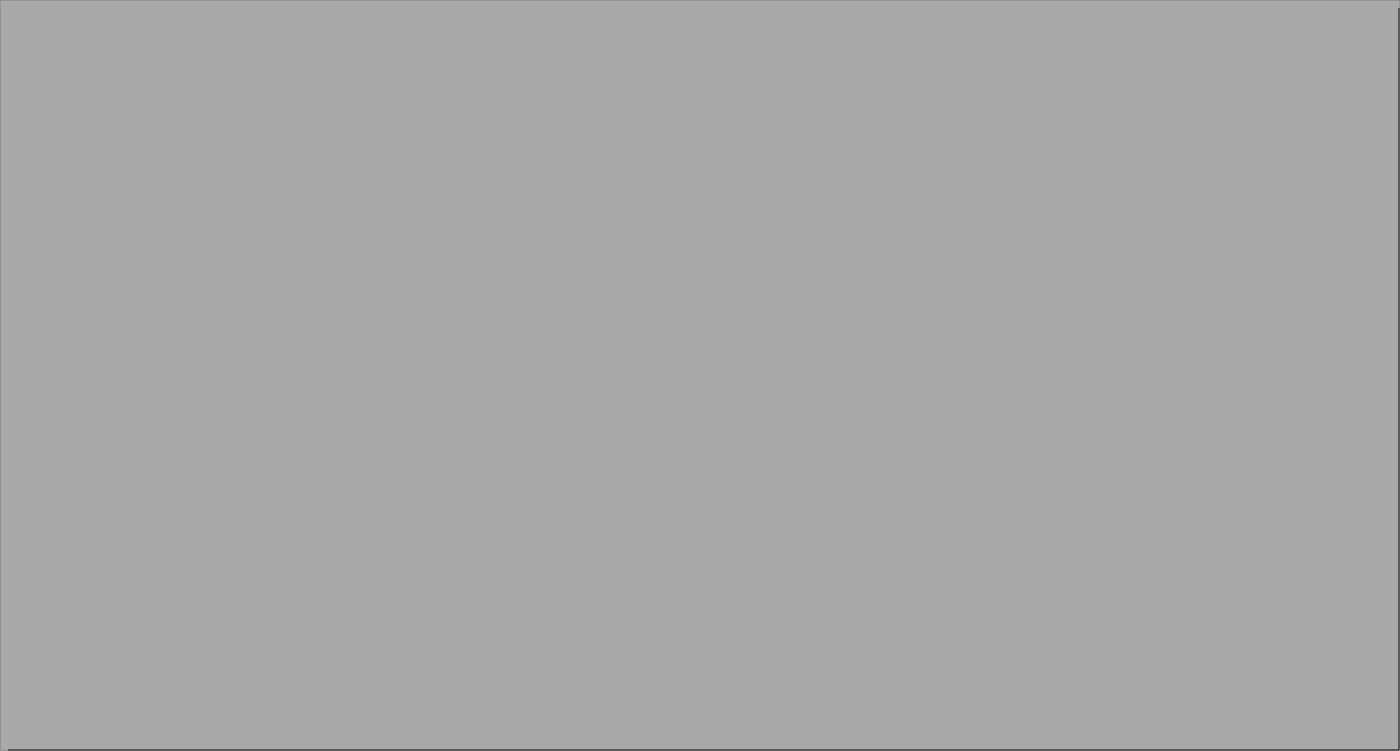
VISUALIZATION PID_alt  // 1792x962, background image 
    Rectangle (10,960 1780x2)
    Rectangle (1790,10 2x950)
END_VISUALIZATION

// ---- Visualizations/Layout.TcVIS
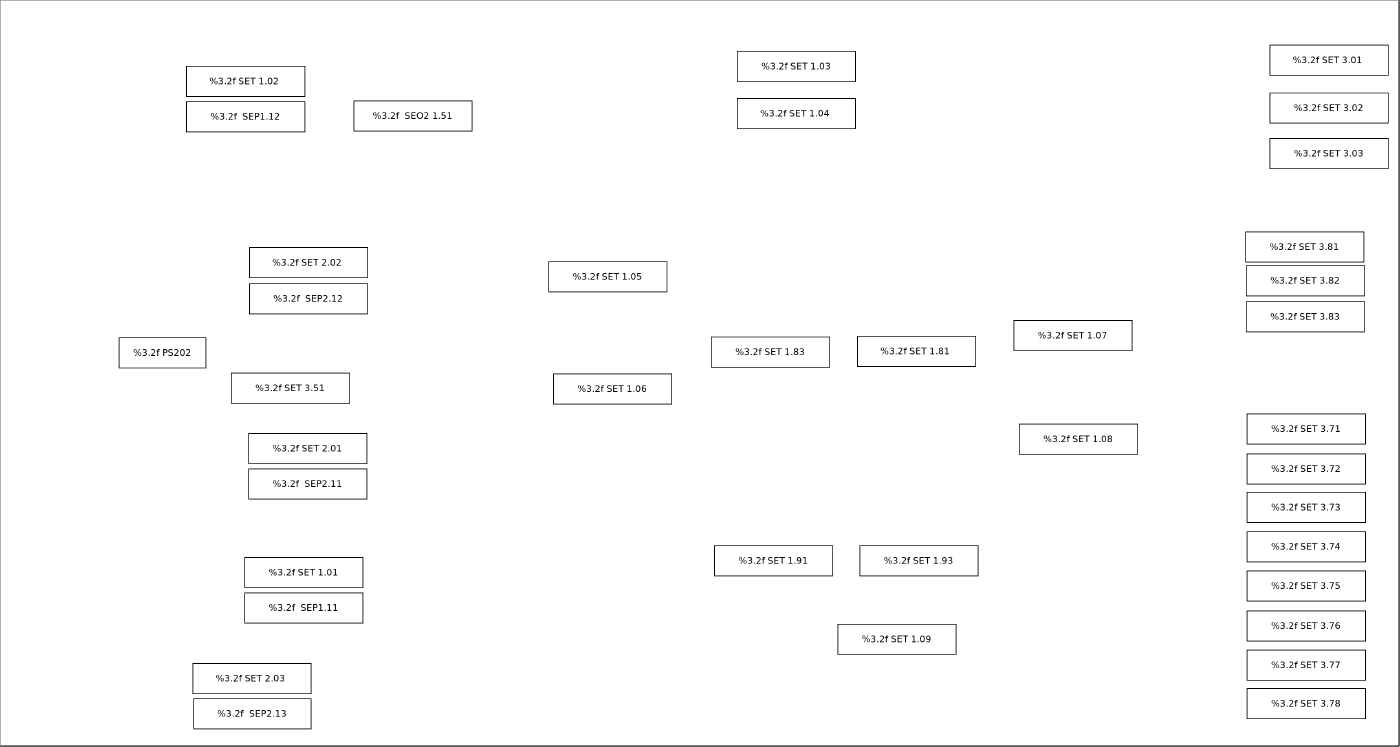
VISUALIZATION Layout  // 1782x952, background image LAyout
    Rectangle (0,950 1780x2)
    Rectangle (1780,0 2x950)
    Rectangle (311,710 151x39), "%3.2f SET 1.01", tooltip "Durchmesser in mm eingeben", text variable: GVL.T_Vor_WT_Visu
    Rectangle (237,84 151x39), "%3.2f SET 1.02", tooltip "Durchmesser in mm eingeben", text variable: GVL.T_nach_WT_Visu
    Rectangle (237,129 151x39), "%3.2f SEP1.12", tooltip "Durchmesser in mm eingeben", text variable: P_nach_WT_Visu
    Rectangle (450,128 151x39), "%3.2f SEO2 1.51", tooltip "Durchmesser in mm eingeben", text variable: GVL.O2_Visu
    Rectangle (317,315 151x39), "%3.2f SET 2.02", tooltip "Durchmesser in mm eingeben", text variable: GVL.T_Komp_Auslass_Visu
    Rectangle (317,361 151x39), "%3.2f SEP2.12", tooltip "Durchmesser in mm eingeben", text variable: GVL.P_Komp_Auslass_Visu
    Rectangle (316,597 151x39), "%3.2f SEP2.11", tooltip "Durchmesser in mm eingeben", text variable: GVL.P_Komp_Einlass_Visu
    Rectangle (294,475 151x39), "%3.2f SET 3.51", tooltip "Durchmesser in mm eingeben", text variable: GVL.T_DK_Steigband3_Visu
    Rectangle (316,552 151x39), "%3.2f SET 2.01", tooltip "Durchmesser in mm eingeben", text variable: GVL.T_Komp_Einlass_Visu
    Rectangle (245,845 151x39), "%3.2f SET 2.03", tooltip "Durchmesser in mm eingeben", text variable: GVL.T_Kond_Auslass_Visu
    Rectangle (311,755 151x39), "%3.2f SEP1.11", tooltip "Durchmesser in mm eingeben", text variable: GVL.P_Vor_WT_Visu
    Rectangle (698,333 151x39), "%3.2f SET 1.05", tooltip "Durchmesser in mm eingeben", text variable: GVL.T_Einduesung_Oben_Visu
    Rectangle (704,476 151x39), "%3.2f SET 1.06", tooltip "Durchmesser in mm eingeben", text variable: GVL.T_Einduesung_Unten_Visu
    Rectangle (938,65 151x39), "%3.2f SET 1.03", tooltip "Durchmesser in mm eingeben", text variable: T_HE_Einduesung_Oben_Visu
    Rectangle (938,125 151x39), "%3.2f SET 1.04", tooltip "Durchmesser in mm eingeben", text variable: T_HE_Einduesung_Unten_Visu
    Rectangle (905,429 151x39), "%3.2f SET 1.83", tooltip "Durchmesser in mm eingeben", text variable: GVL.T_DK_Band_oben3_Visu
    Rectangle (1091,428 151x39), "%3.2f SET 1.81", tooltip "Durchmesser in mm eingeben", text variable: GVL.T_DK_Band_oben1_Visu
    Rectangle (909,695 151x39), "%3.2f SET 1.91", tooltip "Durchmesser in mm eingeben", text variable: GVL.T_DK_Band_unten1_Visu
    Rectangle (1094,695 151x39), "%3.2f SET 1.93", tooltip "Durchmesser in mm eingeben", text variable: GVL.T_DK_Band_unten3_Visu
    Rectangle (1290,408 151x39), "%3.2f SET 1.07", tooltip "Durchmesser in mm eingeben", text variable: GVL.T_Absaugung_Oben_Visu
    Rectangle (1297,540 151x39), "%3.2f SET 1.08", tooltip "Durchmesser in mm eingeben", text variable: GVL.T_Absaugung_Unten_Visu
    Rectangle (1066,795 151x39), "%3.2f SET 1.09", tooltip "Durchmesser in mm eingeben", text variable: GVL.T_Vor_UmdampfLuefter_Visu
    Rectangle (1616,57 151x39), "%3.2f SET 3.01", tooltip "Durchmesser in mm eingeben", text variable: GVL.T_DK_Oben_Visu
    Rectangle (1616,118 151x39), "%3.2f SET 3.02", tooltip "Durchmesser in mm eingeben", text variable: GVL.T_DK_Mitte_Visu
    Rectangle (1616,176 151x39), "%3.2f SET 3.03", tooltip "Durchmesser in mm eingeben", text variable: GVL.T_DK_Unten_Visu
    Rectangle (1587,527 151x39), "%3.2f SET 3.71", tooltip "Durchmesser in mm eingeben", text variable: GVL.T_Mat_Auslass1_Visu
    Rectangle (1587,578 151x39), "%3.2f SET 3.72", tooltip "Durchmesser in mm eingeben", text variable: GVL.T_Mat_Auslass2_Visu
    Rectangle (1587,627 151x39), "%3.2f SET 3.73", tooltip "Durchmesser in mm eingeben", text variable: GVL.T_Mat_Auslass3_Visu
    Rectangle (1587,677 151x39), "%3.2f SET 3.74", tooltip "Durchmesser in mm eingeben", text variable: GVL.T_Mat_Auslass4_Visu
    Rectangle (1587,727 151x39), "%3.2f SET 3.75", tooltip "Durchmesser in mm eingeben", text variable: GVL.T_Mat_Auslass5_Visu
    Rectangle (1587,778 151x39), "%3.2f SET 3.76", tooltip "Durchmesser in mm eingeben", text variable: GVL.T_Mat_Auslass6_Visu
    Rectangle (1587,828 151x39), "%3.2f SET 3.77", tooltip "Durchmesser in mm eingeben", text variable: GVL.T_Mat_Auslass7_Visu
    Rectangle (1587,877 151x39), "%3.2f SET 3.78", tooltip "Durchmesser in mm eingeben", text variable: GVL.T_Mat_Auslass8_Visu
    Rectangle (1585,295 151x39), "%3.2f SET 3.81", tooltip "Durchmesser in mm eingeben", text variable: GVL.T_DK_Steigband1_Visu
    Rectangle (1586,338 151x39), "%3.2f SET 3.82", tooltip "Durchmesser in mm eingeben", text variable: GVL.T_DK_Steigband2_Visu
    Rectangle (1586,384 151x39), "%3.2f SET 3.83", tooltip "Durchmesser in mm eingeben", text variable: GVL.T_DK_Steigband3_Visu
    Rectangle (246,890 150x39), "%3.2f SEP2.13", tooltip "Durchmesser in mm eingeben", text variable: GVL.P_Kond_Auslass_Visu
    Rectangle (151,430 111x39), "%3.2f PS202", tooltip "Durchmesser in mm eingeben", text variable: Ps_202
END_VISUALIZATION

// ---- Visualizations/Heatreg.TcVIS
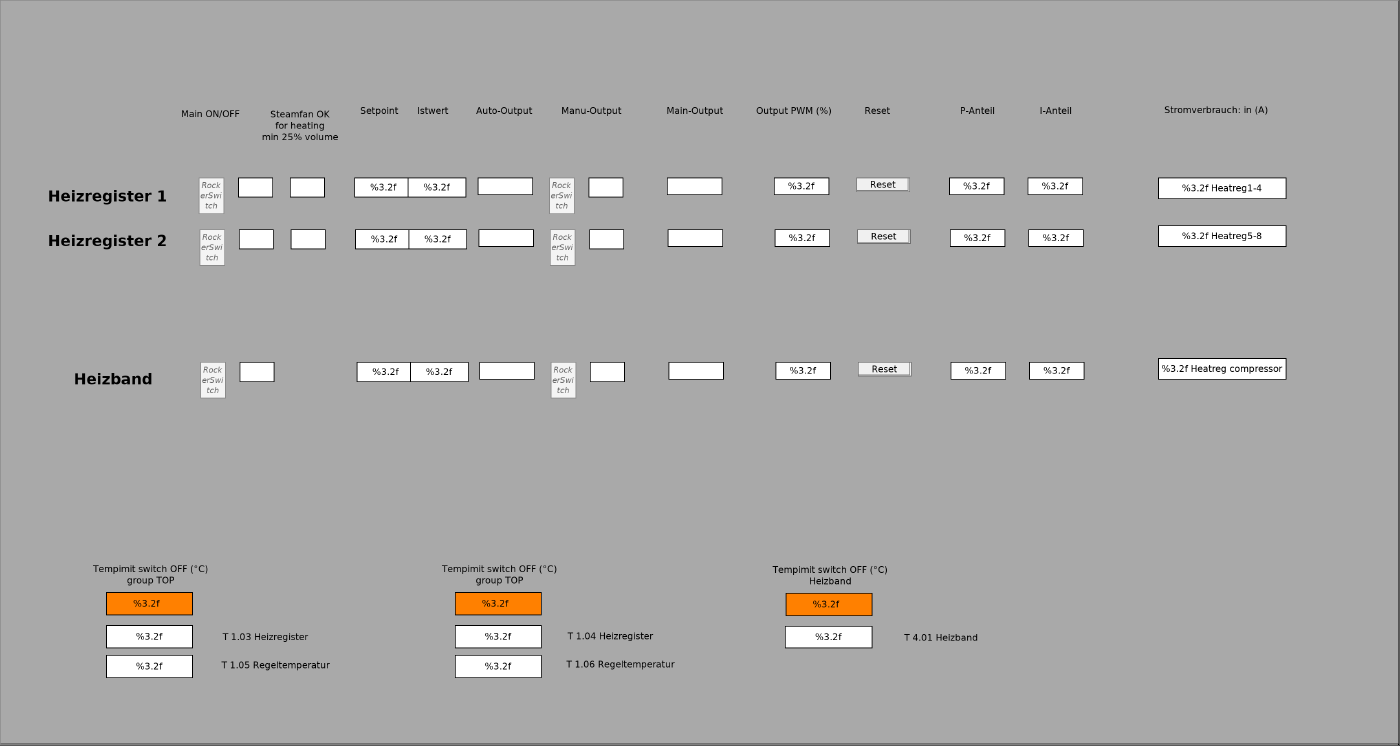
VISUALIZATION Heatreg  // 1782x950
    Rectangle (451,226 74x25), "%3.2f", tooltip "Durchmesser in mm eingeben", text variable: GVL.fSetpointValue1
        OnMouseDown: write the text variable via VisuDialogs.Numpad, min 0, max 150
    Rectangle (596,126 92x30), "Auto-Output"
    Rectangle (707,126 92x30), "Manu-Output"
    Rectangle (839,126 92x30), "Main-Output"
    Rectangle (437,126 92x30), "Setpoint"
    Rectangle (609,292 70x22), colour toggle: GVL.bAuto_Heat_REG2_CTRL
    Rectangle (850,292 70x22), colour toggle: GVL.HEAT_Reg_2_OUT
    Rectangle (608,226 70x22), colour toggle: GVL.bAuto_Heat_REG1_CTRL
    Rectangle (849,226 70x22), colour toggle: GVL.HEAT_Reg_1_OUT
    Rectangle (951,126 116x30), "Output PWM (%)"
    Rectangle (986,292 70x22), "%3.2f", text variable: fPWMDutyCycle2
    Rectangle (985,226 70x22), "%3.2f", text variable: fPWMDutyCycle1
    Rectangle (610,461 70x22), colour toggle: GVL.bAuto_Heat_REG3_CTRL
    Rectangle (851,461 70x22), colour toggle: GVL.HEAT_Reg_3_OUT
    Rectangle (987,461 70x22), "%3.2f", text variable: fPWMDutyCycle3
    Rectangle (1473,124 150x32), "Stromverbrauch: in (A)"
    Rectangle (750,292 44x25), colour toggle: GVL.bManuHeat_REG2_CTRL
    Rectangle (749,226 44x25), colour toggle: GVL.bManuHeat_REG1_CTRL
    Rectangle (751,461 44x25), colour toggle: GVL.bManuHeat_REG3_CTRL
    Rectangle (135,754 110x29), "%3.2f", tooltip "Durchmesser in mm eingeben", text variable: GVL.T_Limit_Heatreg_top
        OnMouseDown: write the text variable via VisuDialogs.Numpad, min 0, max 300
    Rectangle (107,718 170x28), "Tempimit switch OFF (°C) group TOP"
    Rectangle (135,796 110x29), "%3.2f", tooltip "Durchmesser in mm eingeben", text variable: GVL.T_HE_Einduesung_Oben_Visu
    Rectangle (135,834 110x29), "%3.2f", tooltip "Durchmesser in mm eingeben", text variable: GVL.T_Einduesung_Oben_Visu
    Rectangle (265,798 146x26), "T 1.03 Heizregister"
    Rectangle (265,834 172x26), "T 1.05 Regeltemperatur"
    Rectangle (579,754 110x29), "%3.2f", tooltip "Durchmesser in mm eingeben", text variable: GVL.T_Limit_Heatreg_bottom
        OnMouseDown: write the text variable via VisuDialogs.Numpad, min 0, max 300
    Rectangle (551,718 170x28), "Tempimit switch OFF (°C) group TOP"
    Rectangle (579,796 110x29), "%3.2f", tooltip "Durchmesser in mm eingeben", text variable: GVL.T_HE_Einduesung_Unten_Visu
    Rectangle (579,834 110x29), "%3.2f", tooltip "Durchmesser in mm eingeben", text variable: GVL.T_Einduesung_Unten_Visu
    Rectangle (1780,0 2x950)
    Rectangle (0,947 1780x3)
    RockerSwitch (699,226 32x46), variable: GVL.bManuHeat_REG1_CTRL, behaviour: TOGGLE, style: Switch-RockerSwitch-Gray
    RockerSwitch (700,292 32x46), variable: GVL.bManuHeat_REG2_CTRL, behaviour: TOGGLE, style: Switch-RockerSwitch-Gray
    RockerSwitch (701,461 32x46), variable: GVL.bManuHeat_REG3_CTRL, behaviour: TOGGLE, style: Switch-RockerSwitch-Gray
    Rectangle (452,292 74x25), "%3.2f", tooltip "Durchmesser in mm eingeben", text variable: GVL.fSetpointValue2
        OnMouseDown: write the text variable via VisuDialogs.Numpad, min 0, max 150
    Rectangle (454,461 74x25), "%3.2f", tooltip "Durchmesser in mm eingeben", text variable: GVL.fSetpointValue3
        OnMouseDown: write the text variable via VisuDialogs.Numpad, min 0, max 150
    Rectangle (1071,126 92x30), "Reset"
    Button (1092,461 68x18), "Reset"
        tap Reset_heatreg_compressor
    Button (1090,226 68x18), "Reset"
        tap Reset_heatreg_top
    Button (1091,292 68x18), "Reset"
        tap Reset_heatreg_bottom
    Rectangle (370,292 44x25), colour toggle: OK_For_HEAT_WHILE_FAN_IS_ON
    Rectangle (369,226 44x25), colour toggle: OK_For_HEAT_WHILE_FAN_IS_ON
    Rectangle (328,132 108x56), "Steamfan OK for heating min 25% volume"
    Rectangle (304,292 44x25), colour toggle: bManuHeat_REG2_switch_ON
    Rectangle (303,226 44x25), colour toggle: bManuHeat_REG1_switch_ON
    Rectangle (305,461 44x25), colour toggle: bManuHeat_REG3_switch_ON
    RockerSwitch (253,226 32x46), variable: bManuHeat_REG1_switch_ON, behaviour: TOGGLE, style: Switch-RockerSwitch-Gray
    RockerSwitch (254,292 32x46), variable: bManuHeat_REG2_switch_ON, behaviour: TOGGLE, style: Switch-RockerSwitch-Gray
    RockerSwitch (255,461 32x46), variable: bManuHeat_REG3_switch_ON, behaviour: TOGGLE, style: Switch-RockerSwitch-Gray
    Rectangle (222,130 92x30), "Main ON/OFF"
    Rectangle (1198,126 92x30), "P-Anteil"
    Rectangle (1209,292 70x22), "%3.2f", text variable: fKP_Controller_Heatmatt2
        OnMouseDown: write the text variable via VisuDialogs.Numpad, min 0, max 1000
    Rectangle (1208,226 70x22), "%3.2f", text variable: fKP_Controller_Heatmatt1
        OnMouseDown: write the text variable via VisuDialogs.Numpad, min 0, max 1000
    Rectangle (1210,461 70x22), "%3.2f", text variable: fKP_Controller_Heatmatt3
        OnMouseDown: write the text variable via VisuDialogs.Numpad, min 0, max 1000
    Rectangle (1298,126 92x30), "I-Anteil"
    Rectangle (1309,292 70x22), "%3.2f", text variable: fKI_Controller_Heatmatt2
        OnMouseDown: write the text variable via VisuDialogs.Numpad, min 0, max 1000
    Rectangle (1308,226 70x22), "%3.2f", text variable: fKI_Controller_Heatmatt1
        OnMouseDown: write the text variable via VisuDialogs.Numpad, min 0, max 1000
    Rectangle (1310,461 70x22), "%3.2f", text variable: fKI_Controller_Heatmatt3
        OnMouseDown: write the text variable via VisuDialogs.Numpad, min 0, max 1000
    Rectangle (40,235 194x30), "Heizregister 1"
    Rectangle (40,292 194x30), "Heizregister 2"
    Rectangle (47,468 194x30), "Heizband"
    Rectangle (704,797 146x26), "T 1.04 Heizregister"
    Rectangle (704,833 172x26), "T 1.06 Regeltemperatur"
    Rectangle (519,226 74x25), "%3.2f", tooltip "Durchmesser in mm eingeben", text variable: GVL.T_Einduesung_Oben_Visu
    Rectangle (505,126 92x30), "Istwert"
    Rectangle (520,292 74x25), "%3.2f", tooltip "Durchmesser in mm eingeben", text variable: GVL.T_Einduesung_Unten_Visu
    Rectangle (522,461 74x25), "%3.2f", tooltip "Durchmesser in mm eingeben", text variable: T_Komp_Gehaeuse_Visu
    Rectangle (999,797 111x28), "%3.2f", tooltip "Durchmesser in mm eingeben", text variable: T_Komp_Gehaeuse_Visu
    Rectangle (1000,755 110x29), "%3.2f", tooltip "Durchmesser in mm eingeben", text variable: T_Limit_Heatreg3
        OnMouseDown: write the text variable via VisuDialogs.Numpad, min 0, max 300
    Rectangle (972,719 170x28), "Tempimit switch OFF (°C) Heizband"
    Rectangle (1125,799 146x26), "T 4.01 Heizband"
    Rectangle (1474,226 163x27), "%3.2f Heatreg1-4", tooltip "Durchmesser in mm eingeben", text variable: Current_OUT_Heatreg_1_TO_4
    Rectangle (1474,287 163x27), "%3.2f Heatreg5-8", tooltip "Durchmesser in mm eingeben", text variable: Current_OUT_Heatreg_5_TO_8
    Rectangle (1474,456 163x27), "%3.2f Heatreg compressor", tooltip "Durchmesser in mm eingeben", text variable: Current_OUT_Heatreg_Compressor
END_VISUALIZATION

// ---- Visualizations/Sensors.TcVIS
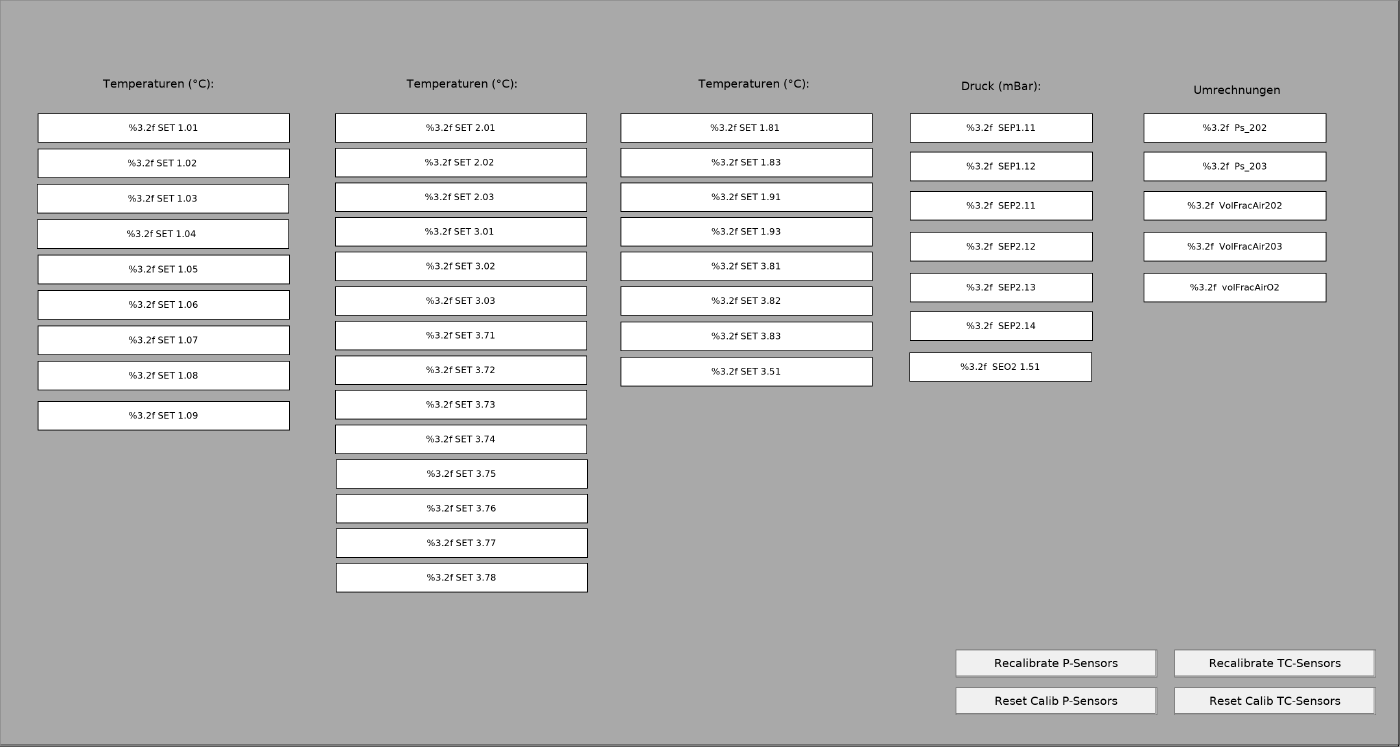
VISUALIZATION Sensors  // 1780x950
    Rectangle (48,144 320x37), "%3.2f SET 1.01", tooltip "Durchmesser in mm eingeben", text variable: GVL.T_Vor_WT_Visu
    Rectangle (48,189 320x37), "%3.2f SET 1.02", tooltip "Durchmesser in mm eingeben", text variable: GVL.T_nach_WT_Visu
    Rectangle (48,324 320x37), "%3.2f SET 1.05", tooltip "Durchmesser in mm eingeben", text variable: GVL.T_Einduesung_Oben_Visu
    Rectangle (48,369 320x37), "%3.2f SET 1.06", tooltip "Durchmesser in mm eingeben", text variable: GVL.T_Einduesung_Unten_Visu
    Rectangle (48,414 320x37), "%3.2f SET 1.07", tooltip "Durchmesser in mm eingeben", text variable: GVL.T_Absaugung_Oben_Visu
    Rectangle (48,459 320x37), "%3.2f SET 1.08", tooltip "Durchmesser in mm eingeben", text variable: GVL.T_Absaugung_Unten_Visu
    Rectangle (48,510 320x37), "%3.2f SET 1.09", tooltip "Durchmesser in mm eingeben", text variable: GVL.T_Vor_UmdampfLuefter_Visu
    Rectangle (120,94 164x25), "Temperaturen (°C):"
    Rectangle (1157,243 232x37), "%3.2f SEP2.11", tooltip "Durchmesser in mm eingeben", text variable: GVL.P_Komp_Einlass_Visu
    Rectangle (1203,97 140x25), "Druck (mBar):"
    Rectangle (1157,295 232x37), "%3.2f SEP2.12", tooltip "Durchmesser in mm eingeben", text variable: GVL.P_Komp_Auslass_Visu
    Rectangle (1157,144 232x37), "%3.2f SEP1.11", tooltip "Durchmesser in mm eingeben", text variable: GVL.P_Vor_WT_Visu
    Rectangle (1156,448 232x37), "%3.2f SEO2 1.51", tooltip "Durchmesser in mm eingeben", text variable: GVL.O2_Visu
    Rectangle (426,144 320x37), "%3.2f SET 2.01", tooltip "Durchmesser in mm eingeben", text variable: GVL.T_Komp_Einlass_Visu
    Rectangle (426,188 320x37), "%3.2f SET 2.02", tooltip "Durchmesser in mm eingeben", text variable: GVL.T_Komp_Auslass_Visu
    Rectangle (426,232 320x37), "%3.2f SET 2.03", tooltip "Durchmesser in mm eingeben", text variable: GVL.T_Kond_Auslass_Visu
    Rectangle (426,276 320x37), "%3.2f SET 3.01", tooltip "Durchmesser in mm eingeben", text variable: GVL.T_DK_Oben_Visu
    Rectangle (426,320 320x37), "%3.2f SET 3.02", tooltip "Durchmesser in mm eingeben", text variable: GVL.T_DK_Mitte_Visu
    Rectangle (426,364 320x37), "%3.2f SET 3.03", tooltip "Durchmesser in mm eingeben", text variable: GVL.T_DK_Unten_Visu
    Rectangle (426,408 320x37), "%3.2f SET 3.71", tooltip "Durchmesser in mm eingeben", text variable: GVL.T_Mat_Auslass1_Visu
    Rectangle (426,452 320x37), "%3.2f SET 3.72", tooltip "Durchmesser in mm eingeben", text variable: GVL.T_Mat_Auslass2_Visu
    Rectangle (426,496 320x37), "%3.2f SET 3.73", tooltip "Durchmesser in mm eingeben", text variable: GVL.T_Mat_Auslass3_Visu
    Rectangle (504,94 168x25), "Temperaturen (°C):"
    Rectangle (426,540 320x37), "%3.2f SET 3.74", tooltip "Durchmesser in mm eingeben", text variable: GVL.T_Mat_Auslass4_Visu
    Rectangle (789,144 320x37), "%3.2f SET 1.81", tooltip "Durchmesser in mm eingeben", text variable: GVL.T_DK_Band_oben1_Visu
    Rectangle (789,188 320x37), "%3.2f SET 1.83", tooltip "Durchmesser in mm eingeben", text variable: GVL.T_DK_Band_oben3_Visu
    Rectangle (789,232 320x37), "%3.2f SET 1.91", tooltip "Durchmesser in mm eingeben", text variable: GVL.T_DK_Band_unten1_Visu
    Rectangle (789,276 320x37), "%3.2f SET 1.93", tooltip "Durchmesser in mm eingeben", text variable: GVL.T_DK_Band_unten3_Visu
    Rectangle (789,320 320x37), "%3.2f SET 3.81", tooltip "Durchmesser in mm eingeben", text variable: GVL.T_DK_Steigband1_Visu
    Rectangle (874,94 170x25), "Temperaturen (°C):"
    Rectangle (789,364 320x37), "%3.2f SET 3.82", tooltip "Durchmesser in mm eingeben", text variable: GVL.T_DK_Steigband2_Visu
    Rectangle (789,409 320x37), "%3.2f SET 3.83", tooltip "Durchmesser in mm eingeben", text variable: GVL.T_DK_Steigband3_Visu
    Rectangle (1778,0 2x947)
    Rectangle (0,947 1778x3)
    Rectangle (427,584 320x37), "%3.2f SET 3.75", tooltip "Durchmesser in mm eingeben", text variable: GVL.T_Mat_Auslass5_Visu
    Rectangle (427,628 320x37), "%3.2f SET 3.76", tooltip "Durchmesser in mm eingeben", text variable: GVL.T_Mat_Auslass6_Visu
    Rectangle (427,672 320x37), "%3.2f SET 3.77", tooltip "Durchmesser in mm eingeben", text variable: GVL.T_Mat_Auslass7_Visu
    Rectangle (427,716 320x37), "%3.2f SET 3.78", tooltip "Durchmesser in mm eingeben", text variable: GVL.T_Mat_Auslass8_Visu
    Rectangle (47,234 320x37), "%3.2f SET 1.03", tooltip "Durchmesser in mm eingeben", text variable: T_HE_Einduesung_Oben_Visu
    Rectangle (47,279 320x37), "%3.2f SET 1.04", tooltip "Durchmesser in mm eingeben", text variable: T_HE_Einduesung_Unten_Visu
    Rectangle (1157,193 232x37), "%3.2f SEP1.12", tooltip "Durchmesser in mm eingeben", text variable: P_nach_WT_Visu
    Rectangle (1157,347 232x37), "%3.2f SEP2.13", tooltip "Durchmesser in mm eingeben", text variable: GVL.P_Kond_Auslass_Visu
    Rectangle (789,454 320x37), "%3.2f SET 3.51", tooltip "Durchmesser in mm eingeben", text variable: GVL.T_Komp_Gehaeuse_Visu
    Rectangle (1157,396 232x37), "%3.2f SEP2.14", tooltip "Durchmesser in mm eingeben", text variable: P_Abs_Amb_Visu
    Button (1493,826 256x35), "Recalibrate TC-Sensors", pressed state: GVL.Compressor_Switch_ON_Manu
        tap Re_Calibrate_TC
    Button (1493,874 256x35), "Reset Calib TC-Sensors", pressed state: GVL.Compressor_Switch_ON_Manu
        tap Reset_Calib
    Button (1215,826 256x35), "Recalibrate P-Sensors", pressed state: GVL.Compressor_Switch_ON_Manu
        tap Set_Calib_preasure
    Button (1215,874 256x35), "Reset Calib P-Sensors", pressed state: GVL.Compressor_Switch_ON_Manu
        tap Reset_Calib_preasure
    Rectangle (1454,243 232x37), "%3.2f VolFracAir202", tooltip "Durchmesser in mm eingeben", text variable: volFracAir202
    Rectangle (1454,295 232x37), "%3.2f VolFracAir203", tooltip "Durchmesser in mm eingeben", text variable: volFracAir203
    Rectangle (1454,144 232x37), "%3.2f Ps_202", tooltip "Durchmesser in mm eingeben", text variable: Ps_202
    Rectangle (1454,193 232x37), "%3.2f Ps_203", tooltip "Durchmesser in mm eingeben", text variable: Ps_203
    Rectangle (1454,347 232x37), "%3.2f volFracAirO2", tooltip "Durchmesser in mm eingeben", text variable: volFracAirO2
    Rectangle (1503,102 140x25), "Umrechnungen"
END_VISUALIZATION

// ---- Visualizations/Service.TcVIS
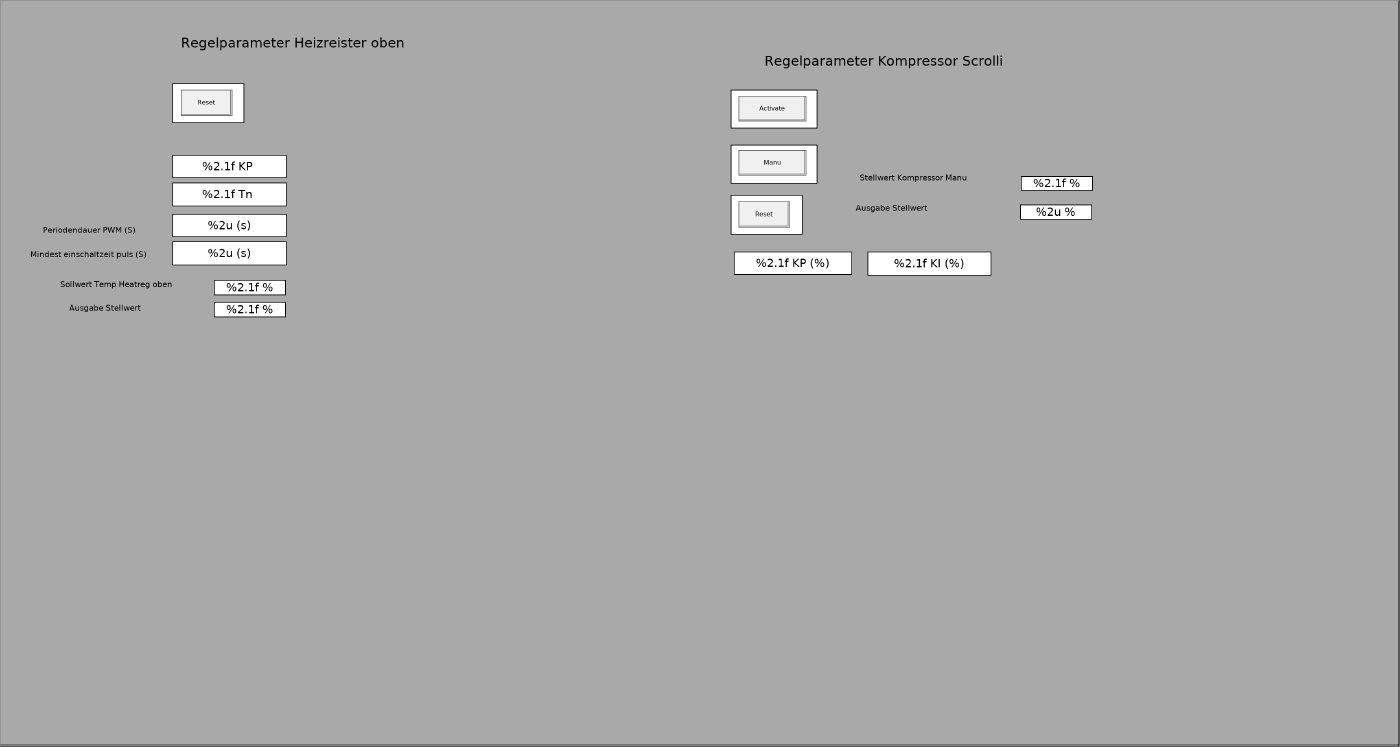
VISUALIZATION Service  // 1780x950
    Rectangle (203,38 339x33), "Regelparameter Heizreister oben"
    Rectangle (272,384 91x19), "%2.1f %", tooltip "Durchmesser in mm eingeben", text variable: fTemp_mean_belt_top
    Rectangle (44,383 179x17), "Ausgabe Stellwert"
    Rectangle (219,106 91x50)
    Button (230,114 65x33), "Reset"
        tap Reset_heatreg_top
    Rectangle (219,197 145x29), "%2.1f KP", tooltip "Durchmesser in mm eingeben", text variable: fKP_Controller_Heatmatt1
        OnMouseDown: write the text variable via VisuDialogs.Numpad, min 0, max 100
    Rectangle (219,232 145x30), "%2.1f Tn", tooltip "Durchmesser in mm eingeben", text variable: fKI_Controller_Heatmatt1
        OnMouseDown: write the text variable via VisuDialogs.Numpad, min 0, max 100
    Rectangle (272,356 91x19), "%2.1f %", tooltip "Durchmesser in mm eingeben", text variable: fSetpointValue1
        OnMouseDown: write the text variable via VisuDialogs.Numpad, min 0, max 100
    Rectangle (29,345 238x33), "Sollwert Temp Heatreg oben"
    Group (919,61 470x289)
        Rectangle (0,0 409x33), "Regelparameter Kompressor Scrolli"
        Rectangle (379,163 91x18), "%2.1f %", tooltip "Durchmesser in mm eingeben", text variable: GVL.fManual_controller_comp
            OnMouseDown: write the text variable via VisuDialogs.Numpad, min 0, max 100
        Rectangle (10,123 110x49), colour toggle: GVL.Set_Manual_controller_comp
        Button (20,130 86x32), "Manu", pressed state: GVL.Set_Manual_controller_comp
            toggle GVL.Set_Manual_controller_comp
        Rectangle (378,199 91x19), "%2u %", tooltip "Durchmesser in mm eingeben", text variable: GVL.fStellwert_comp
        Rectangle (125,195 179x17), "Ausgabe Stellwert"
        Rectangle (10,187 91x50), colour toggle: GVL.Reset_Controller_comp
        Button (20,195 65x33), "Reset"
            tap GVL.Reset_Controller_comp
        Rectangle (14,259 150x29), "%2.1f KP (%)", tooltip "Durchmesser in mm eingeben", text variable: GVL.fKP_Controller_comp
            OnMouseDown: write the text variable via VisuDialogs.Numpad, min 0, max 100
        Rectangle (184,259 157x30), "%2.1f KI (%)", tooltip "Durchmesser in mm eingeben", text variable: GVL.fKI_Controller_comp
            OnMouseDown: write the text variable via VisuDialogs.Numpad, min 0, max 100
        Rectangle (131,156 223x18), "Stellwert Kompressor Manu"
        Rectangle (10,53 110x49), colour toggle: GVL.Activate_controller_comp
        Button (20,61 86x32), "Activate", pressed state: GVL.Activate_controller_comp
            toggle GVL.Activate_controller_comp
    Rectangle (1778,0 2x947)
    Rectangle (0,947 1778x3)
    Rectangle (219,272 145x29), "%2u (s)", tooltip "Durchmesser in mm eingeben", text variable: udiPrd_heatreg1
        OnMouseDown: write the text variable via VisuDialogs.Numpad, min 0, max 100
    Rectangle (219,307 145x30), "%2u (s)", tooltip "Durchmesser in mm eingeben", text variable: udiMinOnTi_heatreg_1
        OnMouseDown: write the text variable via VisuDialogs.Numpad, min 0, max 100
    Rectangle (24,284 179x17), "Periodendauer PWM (S)"
    Rectangle (23,315 179x17), "Mindest einschaltzeit puls (S)"
END_VISUALIZATION

// ---- Visualizations/Farbverlauf.TcVIS
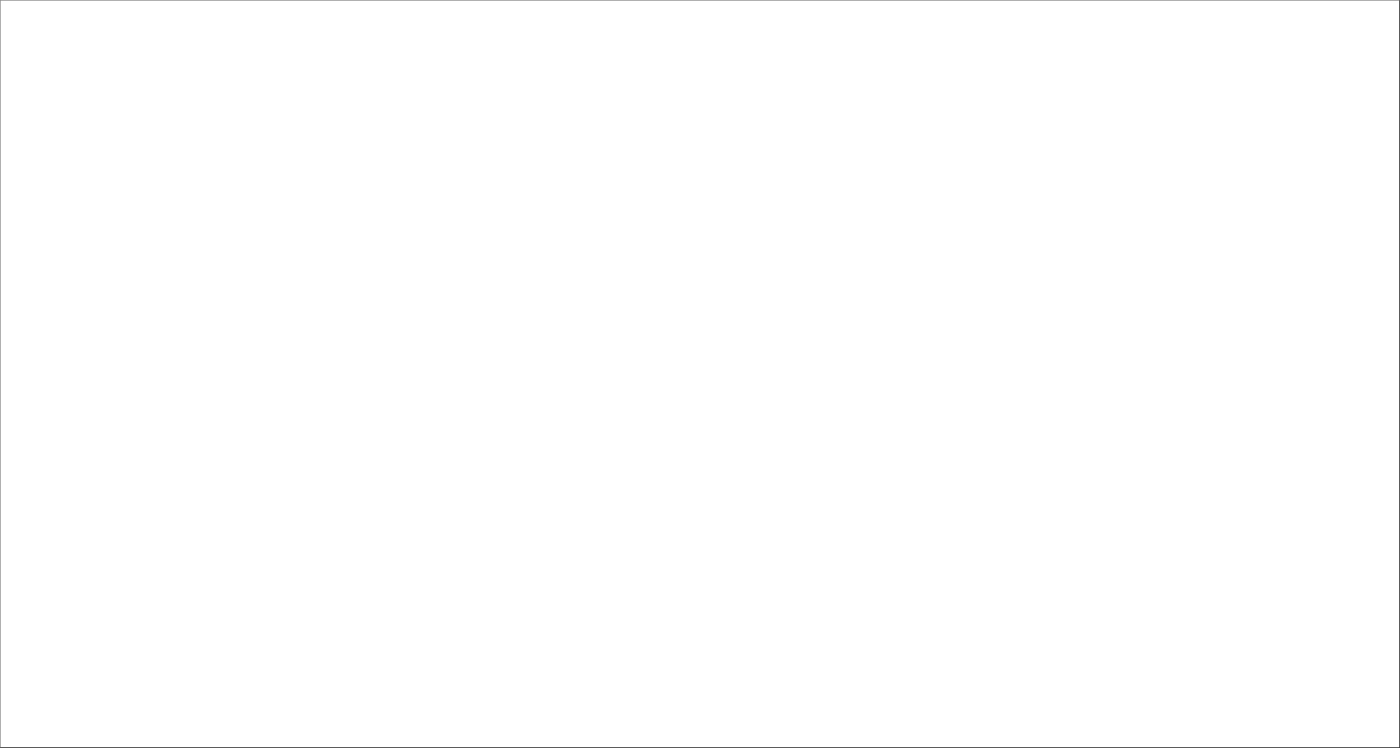
VISUALIZATION Farbverlauf  // 2438x1304
    Rectangle (0,0 2438x1304)
END_VISUALIZATION

// ---- Visualizations/Testseite1.TcVIS
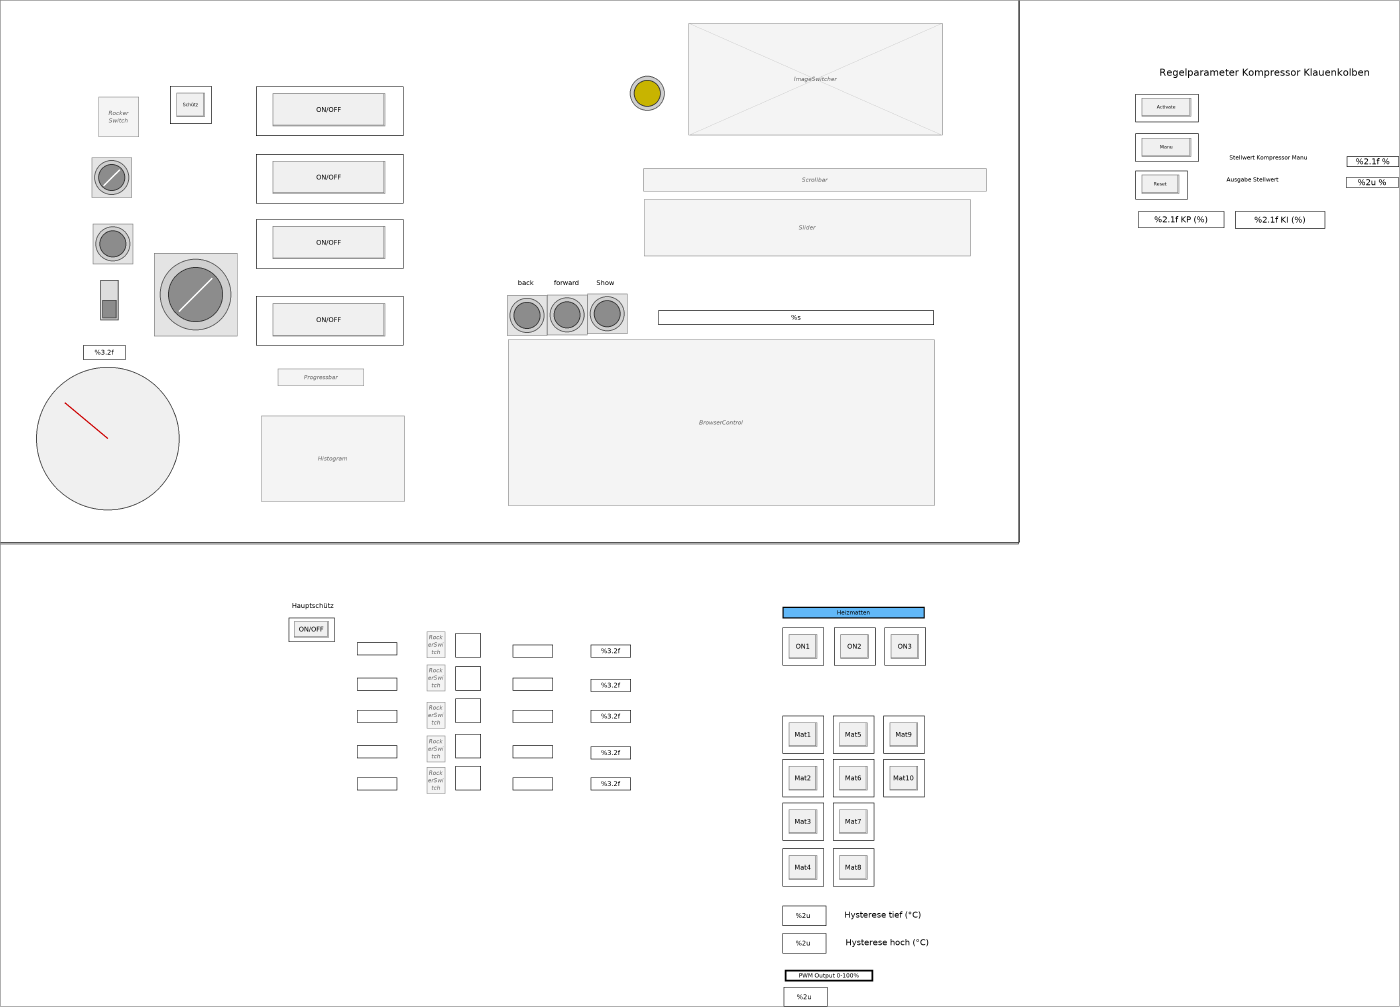
VISUALIZATION Testseite1  // 2444x1759, background image backround
    Rectangle (1778,0 2x947)
    Rectangle (0,947 1778x3)
    PushSwitchLed (162,391 70x70), variable: GVL.bManuHeat_REG3_CTRL, behaviour: TOGGLE, style: Switch-PushSwitchLed-Gray
    RockerSwitch (172,169 70x70), variable: GVL.bManuHeat_REG1_CTRL, behaviour: TOGGLE, style: Switch-RockerSwitch-Gray
    RotarySwitch (160,275 70x70), variable: GVL.bManuHeat_REG2_CTRL, behaviour: TOGGLE, style: Switch-RotarySwitch-Gray
    DipSwitch (156,489 70x70), variable: GVL.bManuHeat_REG4_CTRL, behaviour: TAP, style: Switch-DipSwitch-Gray
    Rectangle (447,269 257x86), colour toggle: GVL.bManuHeat_REG2_CTRL
    Button (476,281 196x57), "ON/OFF", pressed state: GVL.bManuHeat_REG2_CTRL
        toggle GVL.bManuHeat_REG2_CTRL
    Rectangle (447,151 257x86), colour toggle: GVL.bManuHeat_REG1_CTRL
    Button (476,163 196x57), "ON/OFF", pressed state: GVL.bManuHeat_REG1_CTRL
        toggle GVL.bManuHeat_REG1_CTRL
    Rectangle (447,383 257x86), colour toggle: GVL.bManuHeat_REG3_CTRL
    Button (476,395 196x57), "ON/OFF", pressed state: GVL.bManuHeat_REG3_CTRL
        toggle GVL.bManuHeat_REG3_CTRL
    Rectangle (447,517 257x86), colour toggle: GVL.bManuHeat_REG4_CTRL
    Button (476,530 196x57), "ON/OFF", pressed state: GVL.bManuHeat_REG4_CTRL
        toggle GVL.bManuHeat_REG4_CTRL
    Lamp1 (1095,128 70x70), style: Lamp-Lamp1-Yellow
    BrowserControl (887,593 744x290)
        p3734058945: SurlAdress
        p2179181546: bShow
        p2928617338: bBack
        p728663958: bForward
    PushSwitchLed (885,516 70x70), variable: bForward, behaviour: TAP, style: Switch-PushSwitchLed-Gray
    PushSwitchLed (955,515 70x70), variable: bBack, behaviour: TAP, style: Switch-PushSwitchLed-Gray
    PushSwitchLed (1025,513 70x70), variable: bShow, behaviour: TAP, style: Switch-PushSwitchLed-Gray
    Rectangle (886,479 64x30), "back"
    Rectangle (957,479 64x30), "forward"
    Rectangle (1025,479 64x30), "Show"
    Rectangle (1149,542 481x25), "%s", tooltip "Durchmesser in mm eingeben", text variable: SurlAdress
        OnMouseDown: write the text variable via Edit, min 0, max 150
    Histogram (456,726 250x150), scale format: %.1f, scale 0..100
        p1518820177: aArray_Histogram
        p102497268: aArray_Histogram
        p788070771: ARRAY [0..100] OF INT
    Meter360 (63,641 250x250), value: Istwert_IN_NV_OUT, style: Meter-Meter360-Gray, scale format: %.1f, scale 0..100
    Rectangle (145,603 74x25), "%3.2f", tooltip "Durchmesser in mm eingeben", text variable: GVL.fSetpointValue1
        OnMouseDown: write the text variable via VisuDialogs.Numpad, min 0, max 150
    Slider (1124,348 570x99), variable: GVL.fSetpointValue1, scale 0..100
    Scrollbar (1123,294 599x40)
        p1057716461: GVL.fSetpointValue1
    Progressbar (485,644 150x30)
    Potentiometer360 (269,429 145x171), variable: GVL.fSetpointValue1, style: Potentiometer-Potentiometer360-Gray, scale format: %.1f, scale 0..100
        p2431819421: Outside
    Group (623,1103 478x283)
        Rectangle (0,81 70x22), colour toggle: GVL.bAuto_Heat_REG5_CTRL
        Rectangle (272,81 70x22), colour toggle: GVL.HEAT_Reg_5_OUT
        Rectangle (0,19 70x22), colour toggle: GVL.bAuto_Heat_REG4_CTRL
        Rectangle (272,23 70x22), colour toggle: GVL.HEAT_Reg_4_OUT
        Rectangle (408,83 70x22), "%3.2f", text variable: GVL.fPWMDutyCycle5
        Rectangle (408,23 70x22), "%3.2f", text variable: GVL.fPWMDutyCycle4
        Rectangle (0,137 70x22), colour toggle: GVL.bAuto_Heat_REG6_CTRL
        Rectangle (272,137 70x22), colour toggle: GVL.HEAT_Reg_6_OUT
        Rectangle (408,137 70x22), "%3.2f", text variable: GVL.fPWMDutyCycle6
        Rectangle (0,199 70x22), colour toggle: GVL.bAuto_Heat_REG7_CTRL
        Rectangle (272,199 70x22), colour toggle: GVL.HEAT_Reg_7_OUT
        Rectangle (408,201 70x22), "%3.2f", text variable: GVL.fPWMDutyCycle7
        Rectangle (0,255 70x22), colour toggle: GVL.bAuto_Heat_REG8_CTRL
        Rectangle (172,61 44x42), colour toggle: GVL.bManuHeat_REG5_CTRL
        Rectangle (172,3 44x42), colour toggle: GVL.bManuHeat_REG4_CTRL
        Rectangle (172,117 44x42), colour toggle: GVL.bManuHeat_REG6_CTRL
        Rectangle (172,179 44x42), colour toggle: GVL.bManuHeat_REG7_CTRL
        Rectangle (172,235 44x42), colour toggle: GVL.bManuHeat_REG8_CTRL
        Rectangle (272,255 70x22), colour toggle: GVL.HEAT_Reg_8_OUT
        Rectangle (408,255 70x22), "%3.2f", text variable: GVL.fPWMDutyCycle8
        RockerSwitch (122,0 32x46), variable: GVL.bManuHeat_REG4_CTRL, behaviour: TOGGLE, style: Switch-RockerSwitch-Gray
        RockerSwitch (122,58 32x46), variable: GVL.bManuHeat_REG5_CTRL, behaviour: TOGGLE, style: Switch-RockerSwitch-Gray
        RockerSwitch (122,123 32x46), variable: GVL.bManuHeat_REG6_CTRL, behaviour: TOGGLE, style: Switch-RockerSwitch-Gray
        RockerSwitch (122,182 32x46), variable: GVL.bManuHeat_REG7_CTRL, behaviour: TOGGLE, style: Switch-RockerSwitch-Gray
        RockerSwitch (122,237 32x46), variable: GVL.bManuHeat_REG8_CTRL, behaviour: TOGGLE, style: Switch-RockerSwitch-Gray
    Rectangle (504,1079 80x42), colour toggle: GVL.HEAT_Reg_Mainswitch_OUT
    Button (513,1085 61x28), "ON/OFF", pressed state: GVL.HEAT_Reg_Mainswitch_Manu
        toggle GVL.HEAT_Reg_Mainswitch_Manu
    Rectangle (500,1043 92x30), "Hauptschütz"
    Group (1366,1060 270x699)
        Rectangle (0,190 72x66), colour toggle: GVL.Heat_matt1
        Button (11,202 49x42), "Mat1", pressed state: GVL.Heat_matt1_manu
            toggle GVL.Heat_matt1_manu
        Rectangle (88,266 72x66), colour toggle: GVL.Heat_matt6
        Button (99,278 49x42), "Mat6", pressed state: GVL.Heat_matt6_manu
            toggle GVL.Heat_matt6_manu
        Rectangle (0,266 72x66), colour toggle: GVL.Heat_matt2
        Button (11,278 49x42), "Mat2", pressed state: GVL.Heat_matt2_manu
            toggle GVL.Heat_matt2_manu
        Rectangle (88,342 72x66), colour toggle: GVL.Heat_matt7
        Button (99,354 49x42), "Mat7", pressed state: GVL.Heat_matt7_manu
            toggle GVL.Heat_matt7_manu
        Rectangle (0,342 72x66), colour toggle: GVL.Heat_matt3
        Button (11,354 49x42), "Mat3", pressed state: GVL.Heat_matt3_manu
            toggle GVL.Heat_matt3_manu
        Rectangle (88,422 72x66), colour toggle: GVL.Heat_matt8
        Button (99,434 49x42), "Mat8", pressed state: GVL.Heat_matt8_manu
            toggle GVL.Heat_matt8_manu
        Rectangle (0,422 72x66), colour toggle: GVL.Heat_matt4
        Button (11,434 49x42), "Mat4", pressed state: GVL.Heat_matt4_manu
            toggle GVL.Heat_matt4_manu
        Rectangle (176,190 72x66), colour toggle: GVL.Heat_matt9
        Button (187,202 49x42), "Mat9", pressed state: GVL.Heat_matt9_manu
            toggle GVL.Heat_matt9_manu
        Rectangle (88,190 72x66), colour toggle: GVL.Heat_matt5
        Button (99,202 49x42), "Mat5", pressed state: GVL.Heat_matt5_manu
            toggle GVL.Heat_matt5_manu
        Rectangle (176,266 72x66), colour toggle: GVL.Heat_matt10
        Button (187,278 49x42), "Mat10", pressed state: GVL.Heat_matt10_manu
            toggle GVL.Heat_matt10_manu
        Rectangle (0,0 248x20), "Heizmatten"
        Rectangle (178,36 72x66), colour toggle: GVL.Switch_Heat_group3
        Button (189,48 49x42), "ON3", pressed state: GVL.Switch_Heat_group3
            toggle GVL.Switch_Heat_group3
        Rectangle (90,36 72x66), colour toggle: GVL.Switch_Heat_group2
        Button (101,48 49x42), "ON2", pressed state: GVL.Switch_Heat_group2
            toggle GVL.Switch_Heat_group2
        Rectangle (0,36 72x66), colour toggle: GVL.Switch_Heat_group1
        Button (11,48 49x42), "ON1", pressed state: GVL.Switch_Heat_group1
            toggle GVL.Switch_Heat_group1
        Rectangle (2,664 76x35), "%2u", tooltip "Durchmesser in mm eingeben", text variable: GVL.PWM_duty_cycle
            OnMouseDown: write the text variable via VisuDialogs.Numpad, min 0, max 100
        Rectangle (4,634 154x20), "PWM Output 0-100%"
        Rectangle (0,522 76x35), "%2u", tooltip "Durchmesser in mm eingeben", text variable: GVL.Hyst_low_LIM_Heatmatt
            OnMouseDown: write the text variable via VisuDialogs.Numpad, min 0, max 150
        Rectangle (0,570 76x35), "%2u", tooltip "Durchmesser in mm eingeben", text variable: GVL.Hyst_high_LIM_Heatmatt
            OnMouseDown: write the text variable via VisuDialogs.Numpad, min 0, max 150
        Rectangle (94,522 162x32), "Hysterese tief (°C)"
        Rectangle (96,570 174x32), "Hysterese hoch (°C)"
    Rectangle (297,150 72x66), colour toggle: GVL.M_Belt_Feeder_Switch_ON_Manu
    Button (308,162 49x42), "Schütz", pressed state: GVL.M_Belt_Feeder_Switch_ON_Manu
        toggle GVL.M_Belt_Feeder_Switch_ON_Manu
    Rectangle (1972,110 472x33), "Regelparameter Kompressor Klauenkolben"
    Rectangle (2351,273 91x18), "%2.1f %", tooltip "Durchmesser in mm eingeben", text variable: GVL.fManual_controller_Primaer_comp
        OnMouseDown: write the text variable via VisuDialogs.Numpad, min 0, max 100
    Rectangle (1982,233 110x49), colour toggle: GVL.Set_Manual_controller_Primaer_comp
    Button (1993,241 86x32), "Manu", pressed state: GVL.Set_Manual_controller_Primaer_comp
        toggle GVL.Set_Manual_controller_Primaer_comp
    Rectangle (2350,309 91x19), "%2u %", tooltip "Durchmesser in mm eingeben", text variable: GVL.fStellwert_Primaer_comp
    Rectangle (2097,305 179x17), "Ausgabe Stellwert"
    Rectangle (1982,298 91x50), colour toggle: GVL.Reset_Controller_Primaer_comp
    Button (1993,305 65x33), "Reset"
        tap GVL.Reset_Controller_Primaer_comp
    Rectangle (1987,369 150x29), "%2.1f KP (%)", tooltip "Durchmesser in mm eingeben", text variable: GVL.fKP_Controller_Primaer_comp
        OnMouseDown: write the text variable via VisuDialogs.Numpad, min 0, max 100
    Rectangle (2156,369 157x30), "%2.1f KI (%)", tooltip "Durchmesser in mm eingeben", text variable: GVL.fKI_Controller_Primaer_comp
        OnMouseDown: write the text variable via VisuDialogs.Numpad, min 0, max 100
    Rectangle (2103,266 223x18), "Stellwert Kompressor Manu"
    Rectangle (1982,164 110x49), colour toggle: GVL.Activate_controller_Primaer_comp
    Button (1993,171 86x32), "Activate", pressed state: GVL.Activate_controller_Primaer_comp
        toggle GVL.Activate_controller_Primaer_comp
    ImageSwitcher (1202,40 443x196), background image: Triss_PID_V5, image: AQ, behaviour: TOGGLE
        p3148411668: LAyout
END_VISUALIZATION

// ---- Visualizations/FRAME.TcVIS
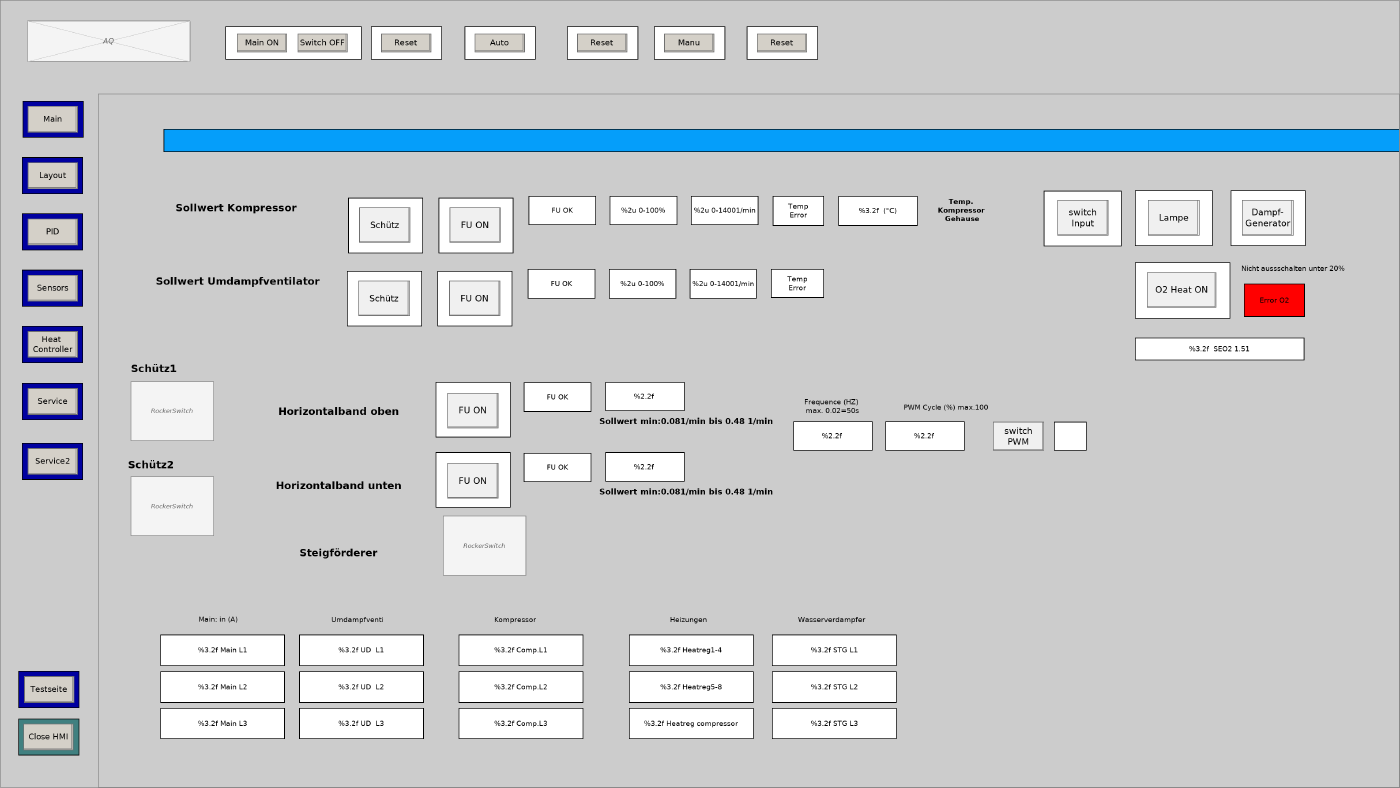
VISUALIZATION FRAME  // 1914x1078
    Frame (134,128 1780x950)
        shows Main()
        shows Heatreg()
        shows Sensors()
        shows Service()
        shows Layout()
        shows PID()
        shows Testseite1()
        shows PID_alt()
    Rectangle (30,215 83x50)
    Rectangle (31,138 83x50)
    Rectangle (30,292 83x50)
    Rectangle (30,369 83x50)
    Rectangle (30,446 83x50)
    Rectangle (30,524 83x50)
    Button (38,145 68x36), "Main"
        OnMouseDown: FrameSelectionChange Selection=SelectedFrame=19e204b9-edb1-49a7-b794-f10e0e8216a7, GlobSel=AssignType=Directly, SelType=Locally
    Rectangle (308,36 186x45), colour toggle: GVL.Mainswitch_OK
    Rectangle (507,36 97x45), colour toggle: GVL.ERROR_Mainswitch
    Rectangle (635,36 97x45), colour toggle: GVL.Control_Auto_active
    Rectangle (775,36 97x45), colour toggle: GVL.Reset_auto
    Rectangle (894,36 97x45), colour toggle: GVL.Control_Manu_active
    Rectangle (1021,36 97x45), colour toggle: GVL.Reset_man
    Button (324,46 68x25), "Main ON"
        tap GVL.Start_Mainswitch
    Button (407,46 68x25), "Switch OFF"
        tap GVL.Switch_OFF_Mainswitch
    Button (521,46 68x25), "Reset"
        tap GVL.RESET_ERROR_Mainswitch
    Button (649,46 68x25), "Auto"
        tap GVL.Control_Auto
    Button (789,46 68x25), "Reset"
        tap GVL.Reset_auto
    Button (908,46 68x25), "Manu"
        tap GVL.Control_Manu
    Button (1035,46 68x25), "Reset"
        tap GVL.Reset_man
    Image (37,28 223x56), image: AQ
    Button (38,222 68x36), "Layout"
        OnMouseDown: FrameSelectionChange Selection=SelectedFrame=19e204b9-edb1-49a7-b794-f10e0e8216a7, Selection=4, GlobSel=AssignType=Directly, SelType=Locally
    Button (38,299 68x36), "PID"
        OnMouseDown: FrameSelectionChange Selection=SelectedFrame=19e204b9-edb1-49a7-b794-f10e0e8216a7, Selection=5, GlobSel=AssignType=Directly, SelType=Locally
    Button (38,376 68x36), "Sensors"
        OnMouseDown: FrameSelectionChange Selection=SelectedFrame=19e204b9-edb1-49a7-b794-f10e0e8216a7, Selection=2, GlobSel=AssignType=Directly, SelType=Locally
    Button (38,453 68x36), "Heat Controller"
        OnMouseDown: FrameSelectionChange Selection=SelectedFrame=19e204b9-edb1-49a7-b794-f10e0e8216a7, Selection=1, GlobSel=AssignType=Directly, SelType=Locally
    Button (38,531 68x36), "Service"
        OnMouseDown: FrameSelectionChange Selection=SelectedFrame=19e204b9-edb1-49a7-b794-f10e0e8216a7, Selection=3, GlobSel=AssignType=Directly, SelType=Locally
    Rectangle (25,983 83x50)
    Button (32,990 68x36), "Close HMI"
        OnMouseDown: FrameSelectionChange Selection=SelectedFrame=19e204b9-edb1-49a7-b794-f10e0e8216a7, Selection=4, GlobSel=AssignType=Directly, SelType=Locally
        OnMouseDown: ExecuteCommand 
        OnMouseDown: CloseDialog Dialog=FileOpenSave, Result=OK, NumpadKeypadSet=True
        OnMouseDown: OpenDialog OpenModal=True, OpenCentered=True
        OnMouseDown: ExecuteCommand 
        OnMouseDown: execute {  }
        OnMouseDown: execute {  }
        OnMouseDown: ExecuteCommand ExecuteCommand=ExecuteCommand=[Command=ExecuteClientProgram, Value='TASKKILL /IM', Value2='Tc3PlcHMI.exe']
    Rectangle (25,918 83x50)
    Button (33,925 68x36), "Testseite"
        OnMouseDown: FrameSelectionChange Selection=SelectedFrame=19e204b9-edb1-49a7-b794-f10e0e8216a7, Selection=6, GlobSel=AssignType=Directly, SelType=Locally
    Rectangle (30,606 83x50)
    Button (38,613 68x36), "Service2"
        OnMouseDown: FrameSelectionChange Selection=SelectedFrame=19e204b9-edb1-49a7-b794-f10e0e8216a7, Selection=7, GlobSel=AssignType=Directly, SelType=Locally
END_VISUALIZATION
